# B&R Automation Studio project NAEUL004C00R13L518F00 (part 57)

#### Local.var
```iecst
(*2020-05-26*)
(**)
(*Local Action, State & Status*)
VAR
	eAct : ePullerPusherAction := PPActIdle;
	eStat : ePullerPusherAction := PPActIdle;
	eMainStatus : eFBStatus := Idle;
	eStatus : eFBStatus := Idle;
	eStatus1 : eFBStatus := Idle;
	eStatus2 : eFBStatus := Idle;
	eStatus3 : eFBStatus := Idle;
	udiStatus : UDINT := 0;
	udiStatus1 : UDINT := 0;
	udiStatus2 : UDINT := 0;
	udiStatus3 : UDINT := 0;
	sStatTxt : STRING[200] := '';
	a_sStatText : ARRAY[0..50] OF STRING[200] := ['Idling','Going Width','Full Homing','Powering On','Powering Off','Homing','Moving Absolute','Moving Relative','Jogging Open','Jogging Close','Jogging Stop','Resetting Axis Error','Stopping','Writing SDO','Background Starting Module OK Check','Background Stopping Module OK Check','Going Width And Power Off','Reset Servo Module Node',33('')];
END_VAR
(**)
(*Local Alarm*)
VAR
	tyAlmData : tyAlmDat;
	tyAlmData1 : tyAlmDat;
	tyAlmData2 : tyAlmDat;
	tyAlmData3 : tyAlmDat;
	a_tyAlmText : ARRAY[10000..10299] OF tyAlmTxt := [(sAlmText:='Axis Move Abnormally By External Force',sRcyText:='Servo Motor Abnormal Operation. Reset And Resume Operation. If The Problem Persists, Please Contact Nutek For A Possible Solution.'),(sAlmText:='CANOpen Communication Error, ModuleOK Not TRUE',sRcyText:='Fail While Read/Write Data. Reset The Error And Resume Operation.'),(sAlmText:='Power On Time Out While Going New Width',sRcyText:='Timeout Expired Before Operation Completed. Reset And Resume Operation.'),(sAlmText:='Homing Time Out While Going New Width',sRcyText:='Timeout Expired Before Operation Completed. Reset And Resume Operation.'),(sAlmText:='Move Absolute Time Out While Going New Width',sRcyText:='Timeout Expired Before Operation Completed. Reset And Resume Operation.'),(sAlmText:='Stop Motion Time Out While Going New Width',sRcyText:='Timeout Expired Before Operation Completed. Reset And Resume Operation.'),(sAlmText:='Axis Error Reset Failed While Going New Width',sRcyText:='Axis Error Reset Failed. Please Retry Again Reset Operation. If The Problem Persists, Please Contact Nutek For A Possible Solution.'),(sAlmText:='Axis Error Occur In Move Absolute While Going New Width',sRcyText:='Servo Motor Abnormal Operation. Reset And Resume Operation. If The Problem Persists, Please Contact Nutek For A Possible Solution.'),(sAlmText:='Axis Error Occur In Homing While Going New Width',sRcyText:='Servo Motor Abnormal Operation. Reset And Resume Operation. If The Problem Persists, Please Contact Nutek For A Possible Solution.'),(sAlmText:='Homing Done But Home Flag Is Not Activated While Going New Width',sRcyText:='Servo Motor Abnormal Operation. Reset And Resume Operation. If The Problem Persists, Please Contact Nutek For A Possible Solution.'),(sAlmText:='Forward Limit Activated In Homing While Going New Width',sRcyText:='Forward Limit Switch Is Activated. Reset The Error By Operate The Motor Backwards.'),(sAlmText:='Reverse Limit Activated In Homing While Going New Width',sRcyText:='Reverse Limit Switch Is Activated. Reset The Error By Operate The Motor Backwards.'),(sAlmText:='Forward Limit Activated In Move Absolute While Going New Width',sRcyText:='Forward Limit Switch Is Activated. Reset The Error By Operate The Motor Backwards.'),(sAlmText:='Reverse Limit Activated In Move Absolute While Going New Width',sRcyText:='Reverse Limit Switch Is Activated. Reset The Error By Operate The Motor Backwards.'),(sAlmText:='Power On Time Out While Full Homing',sRcyText:='Timeout Expired Before Operation Completed. Reset And Resume Operation.'),(sAlmText:='Homing Time Out While Full Homing',sRcyText:='Timeout Expired Before Operation Completed. Reset And Resume Operation.'),(sAlmText:='Stop Motion Time Out While Full Homing',sRcyText:='Timeout Expired Before Operation Completed. Reset And Resume Operation.'),(sAlmText:='Axis Error Reset Failed While Full Homing',sRcyText:='Axis Error Reset Failed. Please Retry Again Reset Operation. If The Problem Persists, Please Contact Nutek For A Possible Solution.'),(sAlmText:='Axis Error Occur In Homing While Full Homing',sRcyText:='Servo Motor Abnormal Operation. Reset And Resume Operation. If The Problem Persists, Please Contact Nutek For A Possible Solution.'),(sAlmText:='Homing Done But Home Flag Is Not Activated While Full Homing',sRcyText:='Servo Motor Abnormal Operation. Reset And Resume Operation. If The Problem Persists, Please Contact Nutek For A Possible Solution.'),(sAlmText:='Forward Limit Activated In Homing While Full Homing',sRcyText:='Forward Limit Switch Is Activated. Reset The Error By Operate The Motor Backwards.'),(sAlmText:='Reverse Limit Activated In Homing While Full Homing',sRcyText:='Reverse Limit Switch Is Activated. Reset The Error By Operate The Motor Backwards.'),(sAlmText:='Power On Time Out',sRcyText:='Timeout Expired Before Operation Completed. Reset And Resume Operation.'),(sAlmText:='Power Off Time Out',sRcyText:='Timeout Expired Before Operation Completed. Reset And Resume Operation.'),(sAlmText:='Homing Time Out',sRcyText:='Timeout Expired Before Operation Completed. Reset And Resume Operation.'),(sAlmText:='Move Absolute Time Out',sRcyText:='Timeout Expired Before Operation Completed. Reset And Resume Operation.'),(sAlmText:='Move Relative Time Out',sRcyText:='Timeout Expired Before Operation Completed. Reset And Resume Operation.'),(sAlmText:='Stop Motion Time Out',sRcyText:='Timeout Expired Before Operation Completed. Reset And Resume Operation.'),(sAlmText:='SDO Write Error',sRcyText:='Fail While Write Data. Reset The Error And Resume Operation.'),(sAlmText:='Request Absolute Position Out Of Range',sRcyText:='Request Absolute Position Does Not Fall Within The Expected Range.'),(sAlmText:='Inlet Sensor Interrupt Auto Width Movement',sRcyText:='Operation Stop Due To The Interruption Of Sensor While Auto Width Moving. Solve The Interruption To Resume Operation.'),(sAlmText:='Outlet Sensor Interrupt Auto Width Movement',sRcyText:='Operation Stop Due To The Interruption Of Sensor While Auto Width Moving. Solve The Interruption To Resume Operation.'),(sAlmText:='Clear Sensor Interrupt Auto Width Movement',sRcyText:='Operation Stop Due To The Interruption Of Sensor While Auto Width Moving. Solve The Interruption To Resume Operation.'),(sAlmText:='Middle Sensor Interrupt Auto Width Movement',sRcyText:='Operation Stop Due To The Interruption Of Sensor While Auto Width Moving. Solve The Interruption To Resume Operation.'),(sAlmText:='Sensor Interrupt Auto Width Movement',sRcyText:='Operation Stop Due To The Interruption Of Sensor While Auto Width Moving. Solve The Interruption To Resume Operation.'),(sAlmText:='Power On Time Out While Going New Width And Off',sRcyText:='Timeout Expired Before Operation Completed. Reset And Resume Operation.'),(sAlmText:='Homing Time Out While Going New Width And Off',sRcyText:='Timeout Expired Before Operation Completed. Reset And Resume Operation.'),(sAlmText:='Move Absolute Time Out While Going New Width And Off',sRcyText:='Timeout Expired Before Operation Completed. Reset And Resume Operation.'),(sAlmText:='Stop Motion Time Out While Going New Width And Off',sRcyText:='Timeout Expired Before Operation Completed. Reset And Resume Operation.'),(sAlmText:='Axis Error Reset Failed While Going New Width And Off',sRcyText:='Axis Error Reset Failed. Please Retry Again Reset Operation. If The Problem Persists, Please Contact Nutek For A Possible Solution.'),(sAlmText:='Axis Error Occur In Move Absolute While Going New Width And Off',sRcyText:='Servo Motor Abnormal Operation. Reset And Resume Operation. If The Problem Persists, Please Contact Nutek For A Possible Solution.'),(sAlmText:='Axis Error Occur In Homing While Going New Width And Off',sRcyText:='Servo Motor Abnormal Operation. Reset And Resume Operation. If The Problem Persists, Please Contact Nutek For A Possible Solution.'),(sAlmText:='Homing Done But Home Flag Is Not Activated While Going New Width And Off',sRcyText:='Servo Motor Abnormal Operation. Reset And Resume Operation. If The Problem Persists, Please Contact Nutek For A Possible Solution.'),(sAlmText:='Forward Limit Activated In Homing While Going New Width And Off',sRcyText:='Forward Limit Switch Is Activated. Reset The Error By Operate The Motor Backwards.'),(sAlmText:='Reverse Limit Activated In Homing While Going New Width And Off',sRcyText:='Reverse Limit Switch Is Activated. Reset The Error By Operate The Motor Backwards.'),(sAlmText:='Forward Limit Activated In Move Absolute While Going New Width And Off',sRcyText:='Forward Limit Switch Is Activated. Reset The Error By Operate The Motor Backwards.'),(sAlmText:='Reverse Limit Activated In Move Absolute While Going New Width And Off',sRcyText:='Reverse Limit Switch Is Activated. Reset The Error By Operate The Motor Backwards.'),2((sAlmText:='Sensor Interrupt Auto Width Movement',sRcyText:='Operation Stop Due To The Interruption Of Sensor While Auto Width Moving. Solve The Interruption To Resume Operation.')),249((0)),(sAlmText:='Forward Limit Activated',sRcyText:='Forward Limit Switch Is Activated. Reset The Error By Operate The Motor Backwards.'),(sAlmText:='Reverse Limit Activated',sRcyText:='Reverse Limit Switch Is Activated. Reset The Error By Operate The Motor Backwards.')];
END_VAR
(**)
(*Local Output*)
VAR
	tyParamOut : tyMotionCANParamOut;
	sAxisErrTxt : STRING[80];
	bWidthPosDiff : BOOL;
	bJogOpen : BOOL;
	bJogClose : BOOL;
	bJogging : BOOL;
	bOpenSen : BOOL;
	bCloseSen : BOOL;
END_VAR
(**)
(*Local Input*)
VAR
	udiRstErr : UDINT := 0;
	bPrep : BOOL := TRUE;
	bEn : BOOL := TRUE;
	bDis : BOOL := FALSE;
	bOps : BOOL := FALSE;
	bManual : BOOL := FALSE;
	diWidthAtHmPos : DINT := 400;
	tyTuning : tyMotionCANTuning;
	diGoWidth : DINT := 150;
	diJogVelInUMPS : DINT := 10000;
	diMovePosInUM : DINT := 0;
	diMoveDistInUM : DINT := 0;
	diMoveVelInUMPS : DINT := 10000;
	diMoveAcc : DINT := 500;
	diMoveDec : DINT := 500;
	diMinAbsPosInUM : DINT := -3000;
	diMaxAbsPosInUM : DINT := 10000000;
	diMinWidthInUM : DINT := 70000;
	diMaxWidthInUM : DINT := 460000;
	diWidthOffsetInUM : DINT := 0;
	bInletSensor : BOOL;
	bOutletSensor : BOOL;
	bClearSensor : BOOL;
	bMiddleSensor : BOOL;
	bInterruptSensor : BOOL;
	bOpenInterruptSensor : BOOL;
	bCloseInterruptSensor : BOOL;
	bDir : BOOL;
	bDirBl : BOOL;
	bNoIndexPulse : BOOL;
	usiNode : USINT;
	sDevice : STRING[3];
	sProgNm : STRING[15] := 'AWOpen';
	diMoveBacklashDistInUM : DINT := 3000;
	diPitchInUM : DINT := 3000;
	tyParamInHm : tyMotionCANParamInHm;
	tyParamInConvert : tyMotionCANParamInConvert := (diPitchInUM:=3000);
	bNtSettingsLoadDone : BOOL := TRUE;
	eMotorType : eServoMotorType := DeltaAsdaA2;
	usiJogFwdStep : USINT;
	usiJogRevStep : USINT;
	bJogRevDone : BOOL;
	bJogFwdDone : BOOL;
	bJogStopDone : BOOL;
	bJogFwd : BOOL;
	bJogRev : BOOL;
	diServoTorque : DINT := 100;
	udiMaxTorque : UDINT := 100;
	diRetSpd : DINT := 24000;
END_VAR
(**)
(*Local*)
VAR
	bRstErr : BOOL;
	udiRstErrOld : UDINT;
	bInitDone : BOOL;
	bInitialDone : BOOL;
	bModuleOKChk : BOOL := TRUE;
	bModuleOK : BOOL;
	bModuleNotOK : BOOL := TRUE;
	diMtrPshrExtTrq : DINT := 0;
	bModuleNotOKLock : BOOL;
	bNotInterruptible : BOOL;
	bInterruptSensor1 : BOOL;
	bInterruptSensor2 : BOOL;
	diActualPosInUMOld : DINT;
	diSlowSpeed : DINT := 2800;
	diExtSlowSpeed : DINT := 2800;
	usiRstStep : USINT := 0;
	usiStep : USINT;
	usiCount : USINT;
	fbTm : TON := (PT:=T#2s);
	fbServoModuleNotOk : TON := (IN:=FALSE,PT:=T#2s);
	fbServoModuleOk : TON := (IN:=FALSE,PT:=T#5s);
	fbRstNodeTimer : TON := (PT:=T#3s);
	tyParamInMove : tyMotionCANParamInMove;
	tyParamInDriver : tyMotionCANDriverIn;
	tyParamOutDriver : tyMotionCANDriverOut := (siModOfOpt_6060:=6);
	fbStop : fbMotionCANStop;
	fbRstAxisErr : fbMotionCANRstAxisErr;
	fbJog : fbMotionCANJog;
	fbMovRel : fbMotionCANMovRel;
	fbMovAbs : fbMotionCANMovAbs;
	fbHoming : fbMotionCANHoming;
	fbPwrOff : fbMotionCANPwrOff;
	fbPwrOn : fbMotionCANPwrOn;
	fbFullHm : fbMotionCANFullHm;
	fbFullMovAbs : fbMotionCANFullMovAbs;
	fbFullMovAbsBl : fbMotionCANFullMovAbsBl;
	fbModuleOK : fbMotionCANModuleOK;
	fbSDOWrite : fbCANSDOWriteArrayParam;
	fbSDOWriteTorque : CANopenSDOWrite8;
	udiModuleNum : UDINT := 301;
END_VAR
```

#### Act_Action.st
```iecst
(** 2020-03-16 **)
ACTION Act_Action:

	//Reset Error
	IF (eStatus = Error) AND bRstErr THEN
		p_eAct	:= PPActIdle;
		eStat	:= PPActIdle;

		fMotionCANRstCtrlWord(ADR(tyParamOutDriver));
	END_IF

	//Reset Done
	IF eStatus = Done AND p_eAct = PPActIdle THEN
		eStat	:= PPActIdle;
	END_IF

	//Set p_eAct
	IF (eStatus = Idle
		AND eStatus1 = Idle
		AND eStatus2 = Idle
		AND eStatus3 = Idle)
		OR p_eAct = PPActIdle
		OR p_eAct = PPActStop
		OR (p_eAct = PPActJogStop AND eStatus = Done)
		THEN
		eStat	:= p_eAct;
	END_IF

	IF EDGEPOS(bModuleNotOK) THEN
		eStat := PPActIdle;
	END_IF

END_ACTION
```

#### Act_Alarm.st
```iecst
(** 2020-03-16 **)
ACTION Act_Alarm:

	//Error
	IF EDGEPOS(eStatus = Error) THEN

		tyAlmData.sProgNm		:= p_sProgNm;
		tyAlmData.udiCode		:= udiStatus;
		tyAlmData.eSeverity		:= AlmSeverityError;
		tyAlmData.udiRunTime	:= tyAlmData.udiRunTime + 1;
		tyAlmData.bAlm			:= TRUE;
		tyAlmData.udiModuleNum  := udiModuleNum;
		g_sAWCloseProgNm		:= p_sProgNm;
		//Get Error Message
		IF tyAlmData.udiCode < 10000 OR tyAlmData.udiCode > 10299 THEN
			tyAlmData.sAlmMsg	:= 'Unknown';
			tyAlmData.sRcyMsg	:= 'Unknown';
		ELSE
			tyAlmData.sAlmMsg	:= a_tyAlmText[tyAlmData.udiCode].sAlmText;
			tyAlmData.sRcyMsg	:= a_tyAlmText[tyAlmData.udiCode].sRcyText;
		END_IF

		sStatTxt	:= tyAlmData.sAlmMsg;

	ELSIF bRstErr AND (tyAlmData.udiCode <> 0) THEN

		tyAlmData.udiCode	:= 0;
		tyAlmData.eSeverity	:= AlmSeverityNA;
		tyAlmData.sAlmMsg	:= '';
		tyAlmData.sRcyMsg	:= '';
		tyAlmData.bAlm			:= FALSE;
		sStatTxt	:= a_sStatText[eStat];

	END_IF

END_ACTION
```

#### Act_Alarm1.st
```iecst
(** 2020-03-16 **)
ACTION Act_Alarm1:

	//Error
	IF EDGEPOS(eStatus1 = Error) THEN

		tyAlmData1.sProgNm		:= p_sProgNm;
		tyAlmData1.udiCode		:= udiStatus1;
		tyAlmData1.eSeverity	:= AlmSeverityError;
		tyAlmData1.udiRunTime	:= tyAlmData1.udiRunTime + 1;
		tyAlmData1.bAlm			:= TRUE;
		tyAlmData1.udiModuleNum  := udiModuleNum;
		g_sAWCloseProgNm		:= p_sProgNm;
		//Get Error Message
		IF tyAlmData1.udiCode < 10000 OR tyAlmData1.udiCode > 10099 THEN
			tyAlmData1.sAlmMsg	:= 'Unknown';
			tyAlmData1.sRcyMsg	:= 'Unknown';
		ELSE
			tyAlmData1.sAlmMsg	:= a_tyAlmText[tyAlmData1.udiCode].sAlmText;
			tyAlmData1.sRcyMsg	:= a_tyAlmText[tyAlmData1.udiCode].sRcyText;
		END_IF

		sStatTxt	:= tyAlmData1.sAlmMsg;

	ELSIF bRstErr AND (tyAlmData1.udiCode <> 0) THEN

		tyAlmData1.udiCode		:= 0;
		tyAlmData1.eSeverity	:= AlmSeverityNA;
		tyAlmData1.sAlmMsg		:= '';
		tyAlmData1.sRcyMsg		:= '';
		tyAlmData1.bAlm			:= FALSE;
		sStatTxt	:= a_sStatText[eStat];

	END_IF

END_ACTION
```

#### Act_Alarm2.st
```iecst
(** 2020-03-16 **)
ACTION Act_Alarm2:

	//Error
	IF EDGEPOS(eStatus2 = Error) THEN

		tyAlmData2.sProgNm		:= p_sProgNm;
		tyAlmData2.udiCode		:= udiStatus2;
		tyAlmData2.eSeverity	:= AlmSeverityError;
		tyAlmData2.udiRunTime	:= tyAlmData2.udiRunTime + 1;
		tyAlmData2.bAlm			:= TRUE;
		tyAlmData2.udiModuleNum  := udiModuleNum;
		g_sAWCloseProgNm		:= p_sProgNm;
		//Get Error Message
		IF tyAlmData2.udiCode < 10000 OR tyAlmData2.udiCode > 10099 THEN
			tyAlmData2.sAlmMsg	:= 'Unknown';
			tyAlmData2.sRcyMsg	:= 'Unknown';
		ELSE
			tyAlmData2.sAlmMsg	:= a_tyAlmText[tyAlmData2.udiCode].sAlmText;
			tyAlmData2.sRcyMsg	:= a_tyAlmText[tyAlmData2.udiCode].sRcyText;
		END_IF

		sStatTxt	:= tyAlmData2.sAlmMsg;

	ELSIF bRstErr AND (tyAlmData2.udiCode <> 0) THEN

		tyAlmData2.udiCode		:= 0;
		tyAlmData2.eSeverity	:= AlmSeverityNA;
		tyAlmData2.sAlmMsg		:= '';
		tyAlmData2.sRcyMsg		:= '';
		tyAlmData2.bAlm			:= FALSE;
		sStatTxt	:= a_sStatText[eStat];

	END_IF

END_ACTION
```

#### Act_Alarm3.st
```iecst
(** 2020-03-16 **)
ACTION Act_Alarm3:

	//Error
	IF EDGEPOS(eStatus3 = Error) THEN

		tyAlmData3.sProgNm		:= p_sProgNm;
		tyAlmData3.udiCode		:= udiStatus3;
		tyAlmData3.eSeverity	:= AlmSeverityError;
		tyAlmData3.udiRunTime	:= tyAlmData3.udiRunTime + 1;
		tyAlmData3.bAlm			:= TRUE;
		tyAlmData3.udiModuleNum  := udiModuleNum;
		g_sAWCloseProgNm		:= p_sProgNm;
		//Get Error Message
		IF tyAlmData3.udiCode < 10000 OR tyAlmData3.udiCode > 10099 THEN
			tyAlmData3.sAlmMsg	:= 'Unknown';
			tyAlmData3.sRcyMsg	:= 'Unknown';
		ELSE
			tyAlmData3.sAlmMsg	:= a_tyAlmText[tyAlmData3.udiCode].sAlmText;
			tyAlmData3.sRcyMsg	:= a_tyAlmText[tyAlmData3.udiCode].sRcyText;
		END_IF

		sStatTxt	:= tyAlmData3.sAlmMsg;

	ELSIF bRstErr AND (tyAlmData3.udiCode <> 0) THEN

		tyAlmData3.udiCode		:= 0;
		tyAlmData3.eSeverity	:= AlmSeverityNA;
		tyAlmData3.sAlmMsg		:= '';
		tyAlmData3.sRcyMsg		:= '';
		tyAlmData3.bAlm			:= FALSE;
		sStatTxt	:= a_sStatText[eStat];

	END_IF

END_ACTION
```

#### Act_Background.st
```iecst
(** 2020-05-26 **)
ACTION Act_Background:

	//Update Parameter
	IF bModuleOK = TRUE THEN

		tyParamInMove.diPosInUM		:= p_diMovePosInUM;
		tyParamInMove.diDistInUM	:= p_diMoveDistInUM;
		tyParamInMove.diVelInUMPS	:= p_diMoveVelInUMPS;
		tyParamInMove.diAcc			:= p_diMoveAcc;
		tyParamInMove.diDec			:= p_diMoveDec;

		fMotionCANUpdtDat(ADR(tyParamOut) , p_tyParamInConvert , tyParamOutDriver , tyParamInDriver , tyParamInMove , p_tyParamInHm , p_bDir, p_eNtParamMotorType);

		bWidthPosDiff	:= (tyParamOut.bIsHomed = FALSE) OR ((ABS((fAWWidthToPosInUM(p_diGoWidth , p_diWidthAtHmPos)) - tyParamOut.diActualPosInUM)) > 500);

		p_tyParamInConvert.diPitchInUM	:= fPitchCalc(p_diWidthOffsetInUM , p_diMaxWidthInUM , p_diMinWidthInUM , p_diPitchInUM);

		fbFullMovAbsBl.tyParamInConvert					:= p_tyParamInConvert;

		IF p_bDir = TRUE THEN
			bOpenSen	:= tyParamOut.bFwdLmtSen;
			bCloseSen	:= tyParamOut.bRevLmtSen;
		ELSE
			bOpenSen	:= tyParamOut.bRevLmtSen;
			bCloseSen	:= tyParamOut.bFwdLmtSen;
		END_IF

		CASE p_eNtParamMotorType OF
			DeltaAsdaA2:
				CASE tyParamOut.udiAxisErrID OF
					8976:	sAxisErrTxt	:= 'Over Current';
					12560:	sAxisErrTxt	:= 'Over Voltage';
					12576:	sAxisErrTxt	:= 'Under Voltage';
					12592:	sAxisErrTxt	:= 'Input Power Phase Loss';
					12816:	sAxisErrTxt	:= 'Regeneration Error';
					12848:	sAxisErrTxt	:= 'Overload';
					12849:	sAxisErrTxt	:= 'Pre-overload Warning';
					13056:	sAxisErrTxt	:= 'U,V,W Wiring Error';
					16912:	sAxisErrTxt	:= 'IGBT Temperature Error';
					21296:	sAxisErrTxt	:= 'Memory Error';
					21569:	sAxisErrTxt	:= 'Emergency Stop Activated';
					21570:	sAxisErrTxt	:= 'Forward Limit Switch Error';
					21571:	sAxisErrTxt	:= 'Reverse Limit Switch Error';
					21572:	sAxisErrTxt	:= 'Forward Software Limit';
					21573:	sAxisErrTxt	:= 'Reverse Software Limit';
					21760:	sAxisErrTxt	:= 'DSP Firmware Upgrade';
					25088:	sAxisErrTxt	:= 'CANopen SYNC Error';
					25360:	sAxisErrTxt	:= 'CANopen Data Initial Error';
					25376:	sAxisErrTxt	:= 'Adjustment Error';
					28961:	sAxisErrTxt	:= 'Motor Protection Error';
					28962:	sAxisErrTxt	:= 'Motor Error';
					29445:	sAxisErrTxt	:= 'Encoder Error';
					29446:	sAxisErrTxt	:= 'Encoder Output Error';
					29968:	sAxisErrTxt	:= 'Serial Communication Error';
					29984:	sAxisErrTxt	:= 'Serial Communication Time Out';
					33024:	sAxisErrTxt	:= 'CANbus Error (Bus-off)';
					33040:	sAxisErrTxt	:= 'CANopen SDO receive buffer overrun';
					33056:	sAxisErrTxt	:= 'CANbus Error (Warning)';
					33072:	sAxisErrTxt	:= 'Node Guarding or Heartbeat Error';
					33280:	sAxisErrTxt	:= 'CANopen PDO Object Error';
					33792:	sAxisErrTxt	:= 'Over Speed';
					34304:	sAxisErrTxt	:= 'Abnormal Pulse Control Command';
					34320:	sAxisErrTxt	:= 'Full Closed Loop Excessive Deviation';
					34321:	sAxisErrTxt	:= 'Excessive Deviation';
				END_CASE

			SchneiderLexium28:
				CASE tyParamOut.udiAxisErrID OF
					8724:	sAxisErrTxt	:= 'Over Current';
					8976:	sAxisErrTxt	:= 'Motor Overload';
					8977:	sAxisErrTxt	:= 'Drive overload (foldback)';
					9088:	sAxisErrTxt	:= 'Calculated offsets for current sensors out OF range';
					9089:	sAxisErrTxt := 'Motor phase missing';
					9090:	sAxisErrTxt := 'Overcurrent detected at one OF the digital outputs';
					12560:	sAxisErrTxt	:= 'DC Bus Over Voltage';
					12576:	sAxisErrTxt	:= 'DC Bus Under Voltage';
					12672:	sAxisErrTxt	:= 'Braking Resistor Overload';
					12673:	sAxisErrTxt	:= 'Safety function Safe Torque Off (STO) triggered';
					12674:	sAxisErrTxt	:= 'DC bus voltage measurement';
					12675:	sAxisErrTxt	:= 'Missing mains supply, undervoltage mains supply';
					12676:	sAxisErrTxt := 'The encoder supply voltage has dropped under operational value';
					12677:	sAxisErrTxt := 'The multi turn encoder battery voltage has dropped under 3 Vdc';
					12678:	sAxisErrTxt := 'Internal position synchronization error	detected between the multi turn AND the single turn modules';
					12679:	sAxisErrTxt := 'Generic error code of the multi turn module is detected';
					12697:	sAxisErrTxt := 'Braking resistor overload';
					16512:	sAxisErrTxt	:= 'Drive overtemperature (IPM)';
					16513:	sAxisErrTxt	:= 'Drive overtemperature (controller)';
					16534:	sAxisErrTxt := 'Temperature sensor inoperative';
					17168:	sAxisErrTxt	:= 'Power stage overtemperature';
					17280:	sAxisErrTxt := 'The encoder temperature is too high';
					17424:	sAxisErrTxt	:= 'Motor overtemperature';
					21808:	sAxisErrTxt	:= 'System error detected (nonvolatilememory)';
					21893:	sAxisErrTxt	:= 'Error detected in non-volatile memory';
					21889:	sAxisErrTxt	:= 'System error detected (nonvolatile memory)';
					21890:	sAxisErrTxt	:= 'System error detected (CAN power supply)';
					21891:	sAxisErrTxt	:= 'System error detected (selftest)';
					21894:	sAxisErrTxt	:= 'System error detected (NV ACCESS)';
					25472:	sAxisErrTxt	:= 'Target position rejected';
					25985:	sAxisErrTxt	:= 'System error detected(FPGA)';
					28816:	sAxisErrTxt	:= 'System error detected (FPGA does NOT match firmware)';
					28817:	sAxisErrTxt	:= 'Emergency Stop Activated';
					28961:	sAxisErrTxt := 'Motor blocked';
					29080:	sAxisErrTxt := 'Commutation error detected';
					29568:  sAxisErrTxt	:= 'Error detected in communication with motor encoder';
					29574:	sAxisErrTxt	:= 'Drive is not synchronous wit master cycle';
					29581:	sAxisErrTxt := 'System error detected (encoder)';
					29587:	sAxisErrTxt	:= 'Encoder overvoltage or overcurrent';
					29592:	sAxisErrTxt := 'The returned position value are no longer considered valid';
					29593:	sAxisErrTxt := 'The multi turn encoder requires an explicit configuration command';
					30081:	sAxisErrTxt := 'Target position rejected';
					30082:	sAxisErrTxt := 'No target values received via the fieldbus';
					33072:	sAxisErrTxt	:= 'CANopen: Heartbeat error detected';
					33296:	sAxisErrTxt := 'R_PDO is too short';
					33921:	sAxisErrTxt	:= 'Actual Motor Velocity Too High';
					33553:	sAxisErrTxt	:= 'Motor torque too high FOR an excessive period OF time';
					33664:	sAxisErrTxt := 'Unstable current loop';
					33922:	sAxisErrTxt := 'Velocity deviation too high';
					34321:	sAxisErrTxt	:= 'Position deviation too high';
					34432:	sAxisErrTxt := 'Position deviation via signal output function MC_OK';
					34441:	sAxisErrTxt := 'Position deviation too high (following error)';
					61568:	sAxisErrTxt	:= 'Fieldbus: Communication	error detected';
					65282:	sAxisErrTxt	:= 'Not possible to read data of electronic motor nameplate';
					65296:	sAxisErrTxt	:= 'Forward Limit Switch Error';
					65297:	sAxisErrTxt	:= 'Reverse Limit Switch Error';
					65281:	sAxisErrTxt := 'System error detected';
					65298:	sAxisErrTxt	:= 'Forward Software Limit';
					65299:	sAxisErrTxt	:= 'Reverse Software Limit';
					65301:	sAxisErrTxt := 'The encoder firmware cannot operate on the provided hardware';

				END_CASE

			EstunPronet:
				CASE tyParamOut.udiAxisErrID OF
					65281:	sAxisErrTxt	:= 'Parameter breakdown';//A01
					65282:	sAxisErrTxt	:= 'AD shift channels breakdown';
					65283:	sAxisErrTxt	:= 'Overspeed';
					65284:	sAxisErrTxt	:= 'Overload';
					65285:	sAxisErrTxt := 'Position error counteroverflow ';
					65286:	sAxisErrTxt := 'Position error pulse overflow';
					65287:	sAxisErrTxt	:= 'The setting of electronic gear or given pulse frequency is not reasonable';
					65288:	sAxisErrTxt	:= 'The 1st channel of current detection is wrong.';
					65289:	sAxisErrTxt	:= 'The 2nd channel of current detection is wrong.';
					65290:	sAxisErrTxt	:= 'Incremental Encoder is break off.';//A10
					65292:	sAxisErrTxt	:= 'Overcurrent';
					65293:	sAxisErrTxt	:= 'Overvoltage';
					65294:	sAxisErrTxt	:= 'Undervoltage';
					65295:	sAxisErrTxt := 'Bleeder resistor error';
					65296:	sAxisErrTxt := 'Regeneration error';
					65297:	sAxisErrTxt := 'Resolver error';
					65298:	sAxisErrTxt := 'IGBT superheat alarm';
					65299:	sAxisErrTxt := 'Motor overheat alarm';
					65300:	sAxisErrTxt := 'Power line phase shortage';//A20
					65301:	sAxisErrTxt	:= 'Instantaneous power off alarm';
					65302:	sAxisErrTxt	:= 'Motor temperature detection sensor is break off.';
					65303:	sAxisErrTxt := 'Brake overcurrent alarm';//A23
					65305:	sAxisErrTxt := 'Motor power line U overcurrent';//A25
					65306:	sAxisErrTxt := 'Motor power line V overcurrent';//A26
					65307:	sAxisErrTxt := 'Motor power line W overcurrent';//A27
					65322:	sAxisErrTxt	:= 'Servomotor type error';//A42
					65323:	sAxisErrTxt	:= 'Servo drive type error';
					65325:	sAxisErrTxt	:= 'Absolute encoder multiturn information error';
					65326:	sAxisErrTxt	:= 'Absolute encoder multiturn information overflow';
					65327:	sAxisErrTxt	:= 'Battery voltage below 2.5V';
					65328:	sAxisErrTxt	:= 'Battery voltage below 3.1V';//A48
					65330:	sAxisErrTxt := 'Serial encoder communication overtime ';//A50
					65331:	sAxisErrTxt := 'Absolute encoder overspeed alarm detected';
					65332:  sAxisErrTxt	:= 'Absolute state of serial encoder error';
					65333:	sAxisErrTxt	:= 'Serial encoder calcaution error';
					65334:	sAxisErrTxt := 'Parity bit or end bit in serial encoder control domain error';
					65335:	sAxisErrTxt	:= 'Serial encoder communication data checking error';
					65336:	sAxisErrTxt := 'End bit in serial encoder control domain error';
					65338:	sAxisErrTxt := 'Serial encoder data empty';
					65339:	sAxisErrTxt := 'Serial encoder data format error';
					65340:	sAxisErrTxt := 'Communication module not detected ';//A60
					65341:	sAxisErrTxt := 'Communication unsuccessful';
					65342:	sAxisErrTxt := 'Servo drive can not receive the period data of communication module ';
					65343:	sAxisErrTxt := 'Communication module can not receive the servo drive response data.';
					65344:	sAxisErrTxt := 'Communication module and bus connectionless';
					65346:	sAxisErrTxt := 'CAN communication abnormal';
					65347:	sAxisErrTxt := 'Receiving heartbeat timeout';
					65349:	sAxisErrTxt := 'Synchronization signal monitoring cycle is longer than setting';
					65362: sAxisErrTxt	:= 'Torque output alarm';
				END_CASE
		END_CASE

	ELSE

		tyParamOut.bAxisErr			:= FALSE;
		tyParamOut.bFwdLmtSen		:= FALSE;
		tyParamOut.bInPos			:= FALSE;
		tyParamOut.bIsHomed			:= FALSE;
		tyParamOut.bPosDiff			:= TRUE;
		tyParamOut.bPwrOn			:= FALSE;
		tyParamOut.bRevLmtSen		:= FALSE;
		tyParamOut.bStopped			:= TRUE;
		tyParamOut.diActualPosInUM	:= 0;
		tyParamOut.diHmAcc			:= 0;
		tyParamOut.diHmSpdForSwitch	:= 0;
		tyParamOut.diHmSpdForZero	:= 0;
		tyParamOut.diProfileAcc		:= 0;
		tyParamOut.diProfileDec		:= 0;
		tyParamOut.udiAxisErrID		:= 0;

		bWidthPosDiff				:= TRUE;

	END_IF

	//Abnormal Movement
//	IF eStatus1 <> Error THEN
//		IF p_bOps = TRUE AND eStatus = Idle THEN
//			IF (ABS(tyParamOut.diActualPosInUM - diActualPosInUMOld) > 2000) AND (ABS(tyParamOut.diActualPosInUM - diActualPosInUMOld) < 10000) THEN
//				eStatus1	:= Error;
//				udiStatus1	:= 10000;	//Axis Move Abnormally By External Force
//
//				fMotionCANRstCtrlWord(ADR(tyParamOutDriver));
//				p_eAct	:= PPActIdle;
//				eStat	:= PPActIdle;
//			END_IF
//		ELSE
//			diActualPosInUMOld	:= tyParamOut.diActualPosInUM;
//		END_IF
//	END_IF

	//Reset Error
	IF (eStatus1 = Error) AND bRstErr THEN
		eStatus1	:= Idle;
		udiStatus1	:= 0;
	END_IF

	//Request Position To Movement Out Of Range
	IF p_bOps
		AND((tyParamInMove.diPosInUM < p_diMinAbsPosInUM) OR (tyParamInMove.diPosInUM > p_diMaxAbsPosInUM))
		AND (eStatus2 <> Error) THEN
		eStatus2	:= Error;
		udiStatus2	:= 10029;	//Request Absolute Position Out Of Range

		fMotionCANRstCtrlWord(ADR(tyParamOutDriver));
		p_eAct	:= PPActIdle;
		eStat	:= PPActIdle;
	END_IF

	//Reset Error
	IF (eStatus2 = Error) AND bRstErr THEN
		eStatus2	:= Idle;
		udiStatus2	:= 0;
	END_IF

	//Sensor Interrupt
	IF (bNotInterruptible = TRUE OR bJogging) AND eStatus3 <> Error THEN

		IF p_bInletSensor = TRUE THEN
			eStatus3	:= Error;
			udiStatus3	:= 10030;	//Inlet Sensor Interrupt Auto Width Movement

			fMotionCANRstCtrlWord(ADR(tyParamOutDriver));
			p_eAct	:= PPActIdle;
			eStat	:= PPActIdle;

		ELSIF p_bOutletSensor = TRUE THEN
			eStatus3	:= Error;
			udiStatus3	:= 10031;	//Outlet Sensor Interrupt Auto Width Movement

			fMotionCANRstCtrlWord(ADR(tyParamOutDriver));
			p_eAct	:= PPActIdle;
			eStat	:= PPActIdle;

		ELSIF p_bClearSensor = TRUE THEN
			eStatus3	:= Error;
			udiStatus3	:= 10032;	//Clear Sensor Interrupt Auto Width Movement

			fMotionCANRstCtrlWord(ADR(tyParamOutDriver));
			p_eAct	:= PPActIdle;
			eStat	:= PPActIdle;

		ELSIF p_bMiddleSensor = TRUE THEN
			eStatus3	:= Error;
			udiStatus3	:= 10033;	//Middle Sensor Interrupt Auto Width Movement

			fMotionCANRstCtrlWord(ADR(tyParamOutDriver));
			p_eAct	:= PPActIdle;
			eStat	:= PPActIdle;

		ELSIF p_bInterruptSensor = TRUE THEN
			eStatus3	:= Error;
			udiStatus3	:= 10034;	//Sensor Interrupt Auto Width Movement

			fMotionCANRstCtrlWord(ADR(tyParamOutDriver));
			p_eAct	:= PPActIdle;
			eStat	:= PPActIdle;

		ELSIF p_bCloseInterruptSensor = TRUE AND bJogOpen = FALSE THEN
			eStatus3	:= Error;
			udiStatus3	:= 10047;	//Sensor Interrupt Auto Width Movement

			fMotionCANRstCtrlWord(ADR(tyParamOutDriver));
			p_eAct	:= PPActIdle;
			eStat	:= PPActIdle;

		ELSIF p_bOpenInterruptSensor = TRUE AND bJogClose = FALSE THEN
			eStatus3	:= Error;
			udiStatus3	:= 10048;	//Sensor Interrupt Auto Width Movement

			fMotionCANRstCtrlWord(ADR(tyParamOutDriver));
			p_eAct	:= PPActIdle;
			eStat	:= PPActIdle;
		END_IF

	END_IF

	//Reset Error
	IF (eStatus3 = Error AND bRstErr)
		OR (p_bOpenInterruptSensor AND eStat = PPActJogClose)
		OR (p_bCloseInterruptSensor AND eStat = PPActJogOpen)
		THEN
		eStatus3	:= Idle;
		udiStatus3	:= 0;
	END_IF

	IF bRstErr THEN
		udiStatus	:= 0;
		bJogging	:= FALSE;
		bJogClose	:= FALSE;
		bJogOpen	:= FALSE;
	END_IF

	fbServoModuleOk(IN:= bModuleOK);
	fbServoModuleNotOk(IN:= bModuleOK = FALSE);
	IF fbServoModuleNotOk.Q AND udiStatus <> 10001 THEN

		bModuleNotOK		:= TRUE;
		bModuleNotOKLock	:= TRUE;
		usiRstStep	:= 0;
		tyParamOutDriver.uiCtrlword_6040	:= 0;
		tyParamOutDriver.siModOfOpt_6060	:= 0;
		tyParamOutDriver.diTargetPos_607A	:= 0;
		tyParamOutDriver.udiMoveSpd_6081	:= 0;
		tyParamOutDriver.siHmMethod_6098	:= 0;
		tyParamOutDriver.diJogVel_60FF		:= 0;

		CASE p_eNtParamMotorType OF

			DeltaAsdaA2:
				fbModuleOK(bModuleOK:= FALSE);
				IF eStatus = Idle THEN
					eAct	:= PPActRstNode;
				END_IF

				IF (eStatus = Done OR eStatus = Error)AND eStat = PPActRstNode THEN

					eAct	:= PPActIdle;
				END_IF

			EstunPronet:
				fbModuleOK(bModuleOK:= FALSE);
				IF eStatus = Idle THEN
					eAct	:= PPActRstNode;
				END_IF

				IF (eStatus = Done OR eStatus = Error)AND eStat = PPActRstNode THEN

					eAct	:= PPActIdle;
				END_IF

			SchneiderLexium28:
			// Do Nothing
		END_CASE

	ELSIF bModuleNotOK = TRUE AND fbServoModuleOk.Q THEN

		CASE usiRstStep OF

			0:
				IF eStatus = Idle THEN
					eAct	:= PPActRstAxisErr;
				END_IF

				IF eStatus = Done AND eStat = PPActRstAxisErr THEN
					eAct	:= PPActIdle;
					usiRstStep	:= 4;
				END_IF

			4: tyParamOutDriver.siModOfOpt_6060 := 1;
				usiRstStep	:= 5;

			5: tyParamOutDriver.siModOfOpt_6060 := 1;
				fbRstNodeTimer(IN:=TRUE);

				IF tyParamInDriver.siModOfOptDisp_6061 = 1 THEN
					usiRstStep	:= 6;
					fbRstNodeTimer(IN:=FALSE);
				ELSIF fbRstNodeTimer.Q THEN
					usiRstStep	:= 8;
					fbRstNodeTimer(IN:=FALSE);
				END_IF

			6: tyParamOutDriver.siModOfOpt_6060 := 6;
				fbRstNodeTimer(IN:=FALSE);
				usiRstStep	:= 7;

			7: tyParamOutDriver.siModOfOpt_6060 := 6;
				fbRstNodeTimer(IN:=TRUE);

				IF tyParamInDriver.siModOfOptDisp_6061 = 6 THEN
					usiRstStep	:= 10;
					fbRstNodeTimer(IN:=FALSE);
				ELSIF fbRstNodeTimer.Q THEN
					usiRstStep	:= 9;
					fbRstNodeTimer(IN:=FALSE);
				END_IF

			8:	fbModuleOK(bEn := TRUE, bModuleOK:= FALSE);
				fbRstNodeTimer(IN:=FALSE);
				usiRstStep	:= 9;

			9:	fbModuleOK(bModuleOK:= FALSE);
				IF eStatus = Idle THEN
					eAct	:=PPActRstNode;
				END_IF

				IF eStatus = Done AND eStat = PPActRstNode THEN
					usiRstStep	:= 0;
					eAct		:= PPActIdle;
				END_IF

			10:IF eStatus = Idle THEN
					eAct	:= PPActRstAxisErr;
				END_IF

				IF eStatus = Done AND eStat = PPActRstAxisErr THEN
					eAct			:= PPActIdle;
					usiRstStep	:= 11;
				END_IF

			11:

				IF eStatus = Idle THEN
					eAct	:= PPActSDOWrite;
				END_IF

				IF eStatus = Done AND eStat = PPActSDOWrite THEN
					eAct			:= PPActIdle;
					usiRstStep	:= 13;

				ELSIF udiStatus = 10028 THEN
					eAct			:= PPActIdle;
					usiRstStep	:= 13;
				END_IF

			13: bModuleNotOK	:= FALSE;
				usiRstStep	:= 0;
		END_CASE
	ELSE
		eAct	:= PPActIdle;

	END_IF

	IF tyParamOut.bPosDiff = FALSE THEN
		tyParamOutDriver.uiCtrlword_6040.4	:= FALSE;
	END_IF

END_ACTION
```

#### Act_InitGlobal.st
```iecst
(** 2019-04-09 **)
ACTION Act_InitGlobal:

	(* Always Change If Project Change *)

	//Pass Data To Link
	p_bLinkOpsRun ACCESS p_OpsRun;
	p_bLinkStartupRun ACCESS p_StartupRun;
	p_bLinkPullConvPullerExtCtrl ACCESS p_PshrConvPshrExtCtrl;
	p_bLinkPullConvPullerRetCtrl ACCESS p_PshrConvPshrRetCtrl;
	p_bLinkDIPullerExtRS ACCESS p_DIPusherExtRS;
	p_bLinkDIPullerRetRS ACCESS p_DIPusherRetRS;
	p_bLinkDIPullerExtSlwRS ACCESS p_DIPusherExtSlwSen;
	p_bLinkDIPullerRetSlwRS ACCESS p_DIPusherRetSlwSen;
	p_dintLinkPullerRetSpd ACCESS p_ProdRcpCurrRcp1MtrPshrExtSpd;
	p_dintLinkPullerRetTrq ACCESS p_ProdRcpCurrRcp1MtrPshrExtTorq;

	p_diLinkProdRcpTrq ACCESS p_ProdRcpCurrRcp1MtrPshrExtTorq;
	p_tyLinkTorqParam ACCESS p_NtParamPPTorqParam;

	//Pass Data To Internal Use
	p_udiRstErr ACCESS p_RstErrReset;
	p_bPrep ACCESS p_NtParamProjServoPullPusherPrep;
	p_bOps ACCESS p_OpsStatusRun;
	p_bManual ACCESS p_UIMnlMod;
	p_tyTuning ACCESS p_NtParamPPTuning;
//	p_diJogVelInUMPS ACCESS p_UIMnlPPJogSpd;
	p_diMovePosInUM ACCESS p_UIMnlPPTargetPos;
	p_diMoveDistInUM ACCESS p_UIMnlPPStepSize;
	p_diMoveAcc ACCESS p_NtParamPPAcc;
	p_diMoveDec ACCESS p_NtParamPPDec;
	p_diWidthOffsetInUM ACCESS p_NtParamWidthOffset;
	p_bDir ACCESS p_NtParamPPDir;
	p_bDirBl ACCESS p_NtParamPPDirBl;
	p_usiNode ACCESS p_NtParamPPNode;
	p_sDevice ACCESS p_NtParamPPDevice;
	p_sProgNm ACCESS p_NtParamPPProgNm;
	p_diMoveBacklashDistInUM ACCESS p_NtParamPPMovBlDistInUM;
	p_diPitchInUM ACCESS p_NtParamPPPitchInUM;
	p_tyParamInHm ACCESS p_NtParamPPParamInHm;
	p_tyParamInConvert ACCESS p_NtParamPPParamInConvert;
	p_bNtSettingsLoadDone ACCESS p_StartupNtSettingsLoadDone;
	p_eNtParamMotorType ACCESS p_NtParamPPMotorType;

	p_bInletShutterCloseRS ACCESS p_DIInShutterCloseRS;
	p_bOutletShutterCloseRS ACCESS p_DIOutShutterCloseRS;
	p_bProjInletShutPrep ACCESS p_NtParamProjInletShutPrep;
	p_bProjOutletShutPrep ACCESS p_NtParamProjOutletShutPrep;
	p_bMagWidthChkSen ACCESS p_DIMagWidthChkSen;

	(* Always Change If Project Change *)

END_ACTION
```

#### Act_Initial.st
```iecst
(** 2020-03-16 **)
ACTION Act_Initial:

	//Initial
	sStatTxt	:= a_sStatText[eStat];

	tyParamInMove.diBacklashDistInUM	:= p_diMoveBacklashDistInUM;
	tyParamInMove.diAcc					:= p_diMoveAcc;
	tyParamInMove.diDec					:= p_diMoveDec;

	//p_tyParamInConvert.diPitchInUM	:= fPitchCalc(p_diWidthOffsetInUM , p_diMaxWidthInUM , p_diMinWidthInUM , p_diPitchInUM);

	fbModuleOK.sDevice	:= p_sDevice;
	fbModuleOK.usiNode	:= p_usiNode;
	fbModuleOK.tDlyTm	:= T#5s;
	fbModuleOK(bEn := FALSE);

	fbSDOWrite.sDevice		:= p_sDevice;
	fbSDOWrite.usiNode		:= p_usiNode;
	fbSDOWrite.eMotorType	:= p_eNtParamMotorType;
	fbSDOWrite(bEn := FALSE);

	fbFullMovAbsBl.p_tyParamOutDriver				:= ADR(tyParamOutDriver);
	fbFullMovAbsBl.tyParamInMove.diBacklashDistInUM	:= p_diMoveBacklashDistInUM;
	fbFullMovAbsBl.tyParamInMove.diAcc				:= p_diMoveAcc;
	fbFullMovAbsBl.tyParamInMove.diDec				:= p_diMoveDec;
	//fbFullMovAbsBl.tyParamInConvert					:= p_tyParamInConvert;
	fbFullMovAbsBl.bDir								:= p_bDir;
	fbFullMovAbsBl.bDirBl							:= p_bDirBl;
	fbFullMovAbsBl.bNoIndexPulse					:= p_bNoIndexPulse;
	fbFullMovAbsBl.eMotorType						:= p_eNtParamMotorType;
	fbFullMovAbsBl(bEn := FALSE);

	fbFullMovAbs.p_tyParamOutDriver					:= ADR(tyParamOutDriver);
	fbFullMovAbs.tyParamInMove.diBacklashDistInUM	:= p_diMoveBacklashDistInUM;
	fbFullMovAbs.tyParamInMove.diAcc				:= p_diMoveAcc;
	fbFullMovAbs.tyParamInMove.diDec				:= p_diMoveDec;
	fbFullMovAbs.tyParamInConvert					:= p_tyParamInConvert;
	fbFullMovAbs.bDir								:= p_bDir;
	fbFullMovAbs.bNoIndexPulse						:= p_bNoIndexPulse;
	fbFullMovAbs.eMotorType							:= p_eNtParamMotorType;
	fbFullMovAbs(bEn := FALSE);

	fbFullHm.p_tyParamOutDriver	:= ADR(tyParamOutDriver);
	fbFullHm.bDir				:= p_bDir;
	fbFullHm.bNoIndexPulse		:= p_bNoIndexPulse;
	fbFullHm.eMotorType			:= p_eNtParamMotorType;
	fbFullHm(bEn := FALSE);

	fbPwrOn.p_tyParamOutDriver	:= ADR(tyParamOutDriver);
	fbPwrOn.eMotorType			:= p_eNtParamMotorType;
	fbPwrOn(bEn := FALSE);

	fbPwrOff.p_tyParamOutDriver	:= ADR(tyParamOutDriver);
	fbPwrOff.eMotorType			:= p_eNtParamMotorType;
	fbPwrOff(bEn := FALSE);

	fbHoming.p_tyParamOutDriver	:= ADR(tyParamOutDriver);
	fbHoming.bDir				:= p_bDir;
	fbHoming.bNoIndexPulse		:= p_bNoIndexPulse;
	fbHoming.eMotorType			:= p_eNtParamMotorType;
	fbHoming(bEn := FALSE);

	fbMovAbs.p_tyParamOutDriver					:= ADR(tyParamOutDriver);
	fbMovAbs.tyParamInMove.diBacklashDistInUM	:= p_diMoveBacklashDistInUM;
	fbMovAbs.tyParamInMove.diAcc				:= p_diMoveAcc;
	fbMovAbs.tyParamInMove.diDec				:= p_diMoveDec;
	fbMovAbs.tyParamInConvert					:= p_tyParamInConvert;
	fbMovAbs.bDir								:= p_bDir;
	fbMovAbs.eMotorType							:= p_eNtParamMotorType;
	fbMovAbs(bEn := FALSE);

	fbMovRel.p_tyParamOutDriver					:= ADR(tyParamOutDriver);
	fbMovRel.tyParamInMove.diBacklashDistInUM	:= p_diMoveBacklashDistInUM;
	fbMovRel.tyParamInMove.diAcc				:= p_diMoveAcc;
	fbMovRel.tyParamInMove.diDec				:= p_diMoveDec;
	fbMovRel.tyParamInConvert					:= p_tyParamInConvert;
	fbMovRel.bDir								:= p_bDir;
	fbMovRel.eMotorType							:= p_eNtParamMotorType;
	fbMovRel(bEn := FALSE);

	fbJog.p_tyParamOutDriver	:= ADR(tyParamOutDriver);
	fbJog.tyParamInConvert		:= p_tyParamInConvert;
	fbJog.eMotorType			:= p_eNtParamMotorType;
	fbJog(bEn := FALSE);

	fbRstAxisErr.p_tyParamOutDriver	:= ADR(tyParamOutDriver);
	fbRstAxisErr(bEn := FALSE);

	fbStop.p_tyParamOutDriver	:= ADR(tyParamOutDriver);
	fbStop(bEn := FALSE);

	fbSDOWriteTorque.pDevice := ADR(p_sDevice);
	fbSDOWriteTorque.node	 := p_usiNode;
	fbSDOWriteTorque.index	 := 16#210C;
	fbSDOWriteTorque.subindex:= 0;
	fbSDOWriteTorque.datalen := 2;
	fbSDOWriteTorque(enable := FALSE);

	bModuleNotOK		:= TRUE;

END_ACTION
```

#### Act_InitLocal.st
```iecst
(** 2020-05-26 **)
ACTION Act_InitLocal:

	//Input Reference Link To Local Variable
	p_eAct ACCESS ADR(eAct);
	p_udiRstErr ACCESS ADR(udiRstErr);
	p_bPrep ACCESS ADR(bPrep);
	p_bEn ACCESS ADR(bEn);
	p_bDis ACCESS ADR(bDis);
	p_bOps ACCESS ADR(bOps);
	p_bManual ACCESS ADR(bManual);
	p_diWidthAtHmPos ACCESS ADR(diWidthAtHmPos);
	p_tyTuning ACCESS ADR(tyTuning);
	p_diGoWidth ACCESS ADR(diGoWidth);
	p_diJogVelInUMPS ACCESS ADR(diJogVelInUMPS);
	p_diMovePosInUM ACCESS ADR(diMovePosInUM);
	p_diMoveDistInUM ACCESS ADR(diMoveDistInUM);
	p_diMoveVelInUMPS ACCESS ADR(diMoveVelInUMPS);
	p_diMoveAcc ACCESS ADR(diMoveAcc);
	p_diMoveDec ACCESS ADR(diMoveDec);
	p_diMinAbsPosInUM ACCESS ADR(diMinAbsPosInUM);
	p_diMaxAbsPosInUM ACCESS ADR(diMaxAbsPosInUM);
	p_diMinWidthInUM ACCESS ADR(diMinWidthInUM);
	p_diMaxWidthInUM ACCESS ADR(diMaxWidthInUM);
	p_diWidthOffsetInUM ACCESS ADR(diWidthOffsetInUM);
	p_bInletSensor ACCESS ADR(bInletSensor);
	p_bOutletSensor ACCESS ADR(bOutletSensor);
	p_bClearSensor ACCESS ADR(bClearSensor);
	p_bMiddleSensor ACCESS ADR(bMiddleSensor);
	p_bInterruptSensor ACCESS ADR(bInterruptSensor);
	p_bOpenInterruptSensor ACCESS ADR(bOpenInterruptSensor);
	p_bCloseInterruptSensor ACCESS ADR(bCloseInterruptSensor);
	p_bDir ACCESS ADR(bDir);
	p_bDirBl ACCESS ADR(bDirBl);
	p_bNoIndexPulse ACCESS ADR(bNoIndexPulse);
	p_usiNode ACCESS ADR(usiNode);
	p_sDevice ACCESS ADR(sDevice);
	p_sProgNm ACCESS ADR(sProgNm);
	p_diMoveBacklashDistInUM ACCESS ADR(diMoveBacklashDistInUM);
	p_diPitchInUM ACCESS ADR(diPitchInUM);
	p_tyParamInHm ACCESS ADR(tyParamInHm);
	p_tyParamInConvert ACCESS ADR(tyParamInConvert);
	p_bNtSettingsLoadDone ACCESS ADR(bNtSettingsLoadDone);
	p_eNtParamMotorType ACCESS ADR(eMotorType);
	p_diServoTorque ACCESS ADR(diServoTorque);

END_ACTION
```

#### Act_Link.st
```iecst
(** 2019-03-29 **)
ACTION Act_Link:

//	IF p_bManual = TRUE THEN
//		p_diMoveVelInUMPS ACCESS p_UIMnlPPNomSpd;
//		p_diJogVelInUMPS ACCESS p_UIMnlPPJogSpd;
//	ELSE
//		p_diMoveVelInUMPS ACCESS p_NtParamAWAutoSpd;
//	END_IF

//	IF p_bProjInletShutPrep = TRUE THEN
//
//		IF p_bInletShutterCloseRS
//			THEN
//			bInterruptSensor1 := TRUE;
//		ELSE
//			bInterruptSensor1 := FALSE;
//		END_IF
//	ELSE
//		bInterruptSensor1 := FALSE;
//	END_IF

//	IF p_bProjOutletShutPrep = TRUE THEN
//		IF p_bOutletShutterCloseRS AND p_eAct = PPActJogOpen
//			THEN
//			bInterruptSensor2 := TRUE;
//		ELSE
//			bInterruptSensor2 := FALSE;
//		END_IF
//	ELSE
//		bInterruptSensor2 := FALSE;
//	END_IF

//	IF usiJogFwdStep = 40 AND p_eAct = PPActJogOpen THEN
//		p_bInterruptSensor	:= NOT p_bMagWidthChkSen;
//	END_IF
//
//	IF usiJogRevStep = 40 AND p_eAct = PPActJogClose THEN
//		p_bInterruptSensor  := NOT p_bMagWidthChkSen;
//	END_IF
//
//	IF p_eAct = PPActIdle OR p_eAct = PPActStop THEN
//		p_bInterruptSensor  := FALSE;
//	END_IF

//	p_bInterruptSensor := bInterruptSensor2 OR bInterruptSensor1;// OR p_bLinkSafetyRelay = FALSE;

END_ACTION
```

#### Act_LinkAction.st
```iecst
(** 2019-10-21 **)
ACTION Act_LinkAction:

//	IF eStatus = Idle THEN
		IF bModuleNotOK THEN
			p_eAct ACCESS ADR(eAct);
		ELSE
			IF p_bLinkStartupRun = TRUE THEN
				p_eAct ACCESS p_StartupServoPPAct;
			ELSIF p_bLinkOpsRun = TRUE OR p_bManual = TRUE THEN
				IF p_bLinkPullConvPullerExtCtrl AND NOT bJogFwdDone
					//AND NOT p_bLinkDIPullerExtRS
					THEN
						bJogStopDone := FALSE;

						CASE usiJogFwdStep OF

							0:

	//						diMtrPshrExtTrq    := 10 + (((p_diLinkProdRcpTrq -10)/10)*444/100);
							diMtrPshrExtTrq    := p_tyLinkTorqParam.usiStartTorque + (((p_diLinkProdRcpTrq -10)/10)*p_tyLinkTorqParam.uiRatio/100);

								IF p_bManual THEN
									memcpy(ADR(fbSDOWriteTorque.data0),p_UIMnlMtrPshrExtTorq,1);
									memcpy(ADR(fbSDOWriteTorque.data1),p_UIMnlMtrPshrExtTorq+1,1);
								ELSE
	//								memcpy(ADR(fbSDOWriteTorque.data0),p_ProdRcpCurrRcp1MtrPshrExtTorq,1);
	//								memcpy(ADR(fbSDOWriteTorque.data1),p_ProdRcpCurrRcp1MtrPshrExtTorq+1,1);

									memcpy(ADR(fbSDOWriteTorque.data0),ADR (diMtrPshrExtTrq),1);
									memcpy(ADR(fbSDOWriteTorque.data1),ADR(diMtrPshrExtTrq)+1,1);
								END_IF

								IF eStat <> PPActIdle THEN
									p_eAct := PPActIdle;
									usiJogFwdStep := 20;
								ELSE
									usiJogFwdStep := 20;
								END_IF

							20:
								fbSDOWriteTorque(enable := TRUE);
								IF fbSDOWriteTorque.status = 65535 THEN
									usiJogFwdStep := 22;
								END_IF

							22:
								fbSDOWriteTorque(enable := TRUE);
								IF fbSDOWriteTorque.status = 0 THEN
									fbSDOWriteTorque(enable := FALSE);
									usiJogFwdStep := 30;
								END_IF

							30:
								IF tyParamOut.bPwrOn = FALSE THEN
									p_eAct := PPActPwrOn;

									IF tyParamOut.bPwrOn THEN
										p_eAct := PPActIdle;
										usiJogFwdStep := 40;
									END_IF
								ELSE
									p_eAct := PPActIdle;
									usiJogFwdStep := 40;

								END_IF

						40:

								p_eAct := PPActJogOpen;

								IF EDGEPOS(p_bLinkDIPullerExtSlwRS) THEN
									p_eAct := PPActIdle;
								END_IF

							IF p_bLinkDIPullerExtSlwRS OR p_bLinkDIPullerExtRS  THEN

									p_diJogVelInUMPS := diExtSlowSpeed;

								ELSE
									IF p_bManual THEN
										p_diJogVelInUMPS ACCESS p_UIMnlPPJogSpd;
									ELSE
										p_diJogVelInUMPS := p_dintLinkPullerRetSpd * 3000;//290000/410000//51250//64062//Extend Speed
									END_IF
								END_IF

							//	IF (eStat = PPActJogOpen AND eMainStatus = Done)
							//		OR p_bLinkDIPullerExtRS
								IF p_bLinkDIPullerExtRS
									THEN
									p_eAct := PPActIdle;
	//								p_eAct := PPActStop;
									p_diJogVelInUMPS := 0;
									usiJogFwdStep := 50;

								END_IF

						50:
							p_eAct := PPActJogStop;
	//						p_eAct := PPActStop;
							p_diJogVelInUMPS := 0;
							IF (eStat = PPActJogStop AND eMainStatus = Done)
								THEN
								p_eAct := PPActIdle;
								usiJogFwdStep := 0;
								bJogFwdDone := TRUE;
							END_IF

						END_CASE

				ELSIF p_bLinkPullConvPullerRetCtrl AND NOT bJogRevDone
					//AND NOT p_bLinkDIPullerRetRS
					THEN

					bJogStopDone := FALSE;
					CASE usiJogRevStep OF

						0:
							memcpy(ADR(fbSDOWriteTorque.data0),ADR(udiMaxTorque),1);
							memcpy(ADR(fbSDOWriteTorque.data1),ADR(udiMaxTorque)+1,1);

							IF eStat <> PPActIdle THEN
								p_eAct := PPActIdle;
								usiJogRevStep := 20;
							ELSE
								usiJogRevStep := 20;
							END_IF

						20:
							fbSDOWriteTorque(enable := TRUE);
							IF fbSDOWriteTorque.status = 65535 THEN
								usiJogRevStep := 22;
							END_IF

						22:
							fbSDOWriteTorque(enable := TRUE);
							IF fbSDOWriteTorque.status = 0 THEN
								fbSDOWriteTorque(enable := FALSE);
								usiJogRevStep := 30;
							END_IF

						30:
							IF tyParamOut.bPwrOn = FALSE THEN
								p_eAct := PPActPwrOn;
								IF tyParamOut.bPwrOn THEN
									p_eAct := PPActIdle;
									usiJogRevStep := 40;
								END_IF
							ELSE
								p_eAct := PPActIdle;
								usiJogRevStep := 40;

							END_IF

						40:
							p_eAct := PPActJogClose;

							IF EDGEPOS(p_bLinkDIPullerRetSlwRS) THEN
								p_eAct := PPActIdle;
							END_IF

						IF p_bLinkDIPullerRetSlwRS OR p_bLinkDIPullerRetRS THEN

								p_diJogVelInUMPS := diSlowSpeed;
							ELSE
								IF p_bManual THEN
									p_diJogVelInUMPS ACCESS p_UIMnlPPJogSpd;
								ELSE
								p_diJogVelInUMPS :=  diRetSpd; //36250 //512500 //410000 //16000
								END_IF

							END_IF

						//	IF (eStat = PPActJogClose AND eMainStatus = Done)
						//		OR p_bLinkDIPullerRetRS
							IF p_bLinkDIPullerRetRS
								THEN
								p_eAct := PPActIdle;

								p_diJogVelInUMPS := 0;
								usiJogRevStep := 50;

							END_IF

						50:
							p_eAct := PPActJogStop;
							p_diJogVelInUMPS := 0;
							IF (eStat = PPActJogStop AND eMainStatus = Done)
							THEN
								p_eAct := PPActIdle;
								usiJogRevStep := 0;
								bJogRevDone := TRUE;
							END_IF

					END_CASE
				ELSE

					IF bJogStopDone = FALSE THEN
						p_eAct := PPActJogStop;
					END_IF

					usiJogFwdStep := 0;
					usiJogRevStep := 0;
					p_diJogVelInUMPS := 0;
					tyParamOutDriver.diJogVel_60FF := 0; // ADDED

					IF eStat = PPActJogStop AND eMainStatus = Done THEN
						p_eAct := PPActIdle;
						bJogStopDone := TRUE;
					END_IF

					IF tyParamInDriver.uiErrCode_603F <> 0 THEN //error 12592
						tyParamOutDriver.uiCtrlword_6040 := 0; //0111 (7)> 1111 (15)
					END_IF
				END_IF
			ELSE

				usiJogFwdStep := 0;
				usiJogRevStep := 0;
				p_diJogVelInUMPS := 0;
				IF eStatus <> Idle THEN
					p_eAct := PPActIdle;
					IF eStat = PPActIdle AND eMainStatus = Done THEN
						p_eAct := PPActIdle;
					END_IF
				END_IF
			END_IF
		END_IF
//	END_IF

	IF EDGENEG(p_bManual) OR EDGENEG(p_bLinkOpsRun) OR EDGENEG(p_bLinkStartupRun) THEN
		tyParamOutDriver.uiCtrlword_6040	:= 0;
	END_IF

	IF (eStat = PPActJogClose AND p_bLinkDIPullerRetRS)
		OR (eStat = PPActJogOpen AND p_bLinkDIPullerExtRS)
		THEN
		p_diJogVelInUMPS := 0;
	END_IF

	IF p_bLinkDIPullerRetRS = FALSE THEN
		bJogRevDone := FALSE;
	END_IF

	IF p_bLinkDIPullerExtRS = FALSE THEN
		bJogFwdDone := FALSE;
	END_IF
	//fbPwrOnDlyTmr
END_ACTION
```

#### Act_Main.st
```iecst
(** 2020-05-26 **)
ACTION Act_Main:

	//Main
IF bModuleNotOK = FALSE THEN

		CASE eStat OF

			PPActIdle:
				IF eStatus <> Idle THEN	//Reset Data
					//Private
					fbStop(bEn := FALSE);
					fbRstAxisErr(bEn := FALSE);
					fbJog(bEn := FALSE);
					fbMovRel(bEn := FALSE);
					fbMovAbs(bEn := FALSE);
					fbHoming(bEn := FALSE);
					fbPwrOff(bEn := FALSE);
					fbPwrOn(bEn := FALSE);
					fbFullHm(bEn := FALSE);
					fbFullMovAbs(bEn := FALSE);
					fbFullMovAbsBl(bEn := FALSE);
					fbSDOWrite(bEn := FALSE);
					fbTm(IN := FALSE);
					usiStep				:= 0;
					usiCount			:= 0;
					bNotInterruptible	:= FALSE;
					tyParamOutDriver.uiCtrlword_6040.7	:= FALSE;
					sStatTxt	:= a_sStatText[eStat];

				END_IF

				eStatus	:= Idle;

				IF EDGENEG(p_bManual) THEN
					fMotionCANRstCtrlWord(ADR(tyParamOutDriver));
				END_IF

			PPActGoWidth:
				IF (eStatus = Idle OR eStatus = Busy) THEN

					eStatus	:= Busy;

					sStatTxt	:= a_sStatText[eStat];

					bNotInterruptible	:= TRUE;

					CASE usiStep OF
						0:	//Wait For Motion Parameter Update
							p_diMovePosInUM	:= fAWWidthToPosInUM(p_diGoWidth , p_diWidthAtHmPos);
							usiStep	:= 1;

						1:	//Check Position Difference
							IF tyParamOut.bPosDiff = TRUE THEN
								usiStep	:= 2;
							ELSE
								eStatus	:= Done;
							END_IF

						2:	//Move
							fbFullMovAbsBl.tyParamInDriver					:= tyParamInDriver;
							fbFullMovAbsBl.tyParamInMove.diPosInUM			:= p_diMovePosInUM;
							fbFullMovAbsBl.tyParamInMove.diDistInUM			:= p_diMoveDistInUM;
							fbFullMovAbsBl.tyParamInMove.diVelInUMPS		:= p_diMoveVelInUMPS;
							fbFullMovAbsBl.tyParamInMove.diAcc				:= p_diMoveAcc;
							fbFullMovAbsBl.tyParamInMove.diDec				:= p_diMoveDec;
							fbFullMovAbsBl.tyParamOut						:= tyParamOut;
							fbFullMovAbsBl(bEn := TRUE);

							IF fbFullMovAbsBl.udiStatus = 0 THEN
								eStatus	:= Done;
							ELSIF fbFullMovAbsBl.udiStatus < 65534 THEN
								eStatus		:= Error;

								IF fbFullMovAbsBl.udiStatus = 1401 THEN
									udiStatus	:= 10002;	//Power On Time Out While Going New Width
								ELSIF fbFullMovAbsBl.udiStatus = 1402 THEN
									udiStatus	:= 10003;	//Homing Time Out While Going New Width
								ELSIF fbFullMovAbsBl.udiStatus = 1403 THEN
									udiStatus	:= 10004;	//Move Absolute Time Out While Going New Width
								ELSIF fbFullMovAbsBl.udiStatus = 1405 THEN
									udiStatus	:= 10005;	//Stop Motion Time Out While Going New Width
								ELSIF fbFullMovAbsBl.udiStatus = 1408 THEN
									udiStatus	:= 10006;	//Axis Error Reset Failed While Going New Width
								ELSIF fbFullMovAbsBl.udiStatus = 1409 THEN
									udiStatus	:= 10007;	//Axis Error Occur In Move Absolute While Going New Width
								ELSIF fbFullMovAbsBl.udiStatus = 1411 THEN
									udiStatus	:= 10008;	//Axis Error Occur In Homing While Going New Width
								ELSIF fbFullMovAbsBl.udiStatus = 1412 THEN
									udiStatus	:= 10009;	//Homing Done But Home Flag Is Not Activated While Going New Width
								ELSIF fbFullMovAbsBl.udiStatus = 1413 THEN
									udiStatus	:= 10010;	//Forward Limit Activated In Homing While Going New Width
								ELSIF fbFullMovAbsBl.udiStatus = 1414 THEN
									udiStatus	:= 10011;	//Reverse Limit Activated In Homing While Going New Width
								ELSIF fbFullMovAbsBl.udiStatus = 1415 THEN
									udiStatus	:= 10012;	//Forward Limit Activated In Move Absolute While Going New Width
								ELSIF fbFullMovAbsBl.udiStatus = 1416 THEN
									udiStatus	:= 10013;	//Reverse Limit Activated In Move Absolute While Going New Width
								ELSE
									udiStatus	:= fbFullMovAbsBl.udiStatus;
								END_IF
							END_IF

					END_CASE

				END_IF

			PPActGoWidthOff:
				IF (eStatus = Idle OR eStatus = Busy) THEN

					eStatus	:= Busy;

					sStatTxt	:= a_sStatText[eStat];

					bNotInterruptible	:= TRUE;

					CASE usiStep OF
						0:	//Wait For Motion Parameter Update
							p_diMovePosInUM	:= fAWWidthToPosInUM(p_diGoWidth , p_diWidthAtHmPos);
							usiStep	:= 1;

						1:	//Check Position Difference
							IF tyParamOut.bPosDiff = TRUE THEN
								usiStep	:= 2;
							ELSE
								eStatus	:= Done;
							END_IF

						2:	//Move
							fbFullMovAbsBl.tyParamInDriver					:= tyParamInDriver;
							fbFullMovAbsBl.tyParamInMove.diPosInUM			:= p_diMovePosInUM;
							fbFullMovAbsBl.tyParamInMove.diDistInUM			:= p_diMoveDistInUM;
							fbFullMovAbsBl.tyParamInMove.diVelInUMPS		:= p_diMoveVelInUMPS;
							fbFullMovAbsBl.tyParamInMove.diAcc				:= p_diMoveAcc;
							fbFullMovAbsBl.tyParamInMove.diDec				:= p_diMoveDec;
							fbFullMovAbsBl.tyParamOut						:= tyParamOut;
							fbFullMovAbsBl(bEn := TRUE);

							IF fbFullMovAbsBl.udiStatus = 0 THEN
								usiStep	:= 3;
							ELSIF fbFullMovAbsBl.udiStatus < 65534 THEN
								eStatus		:= Error;

								IF fbFullMovAbsBl.udiStatus = 1401 THEN
									udiStatus	:= 10035;	//Power On Time Out While Going New Width And Off
								ELSIF fbFullMovAbsBl.udiStatus = 1402 THEN
									udiStatus	:= 10036;	//Homing Time Out While Going New Width And Off
								ELSIF fbFullMovAbsBl.udiStatus = 1403 THEN
									udiStatus	:= 10037;	//Move Absolute Time Out While Going New Width And Off
								ELSIF fbFullMovAbsBl.udiStatus = 1405 THEN
									udiStatus	:= 10038;	//Stop Motion Time Out While Going New Width And Off
								ELSIF fbFullMovAbsBl.udiStatus = 1408 THEN
									udiStatus	:= 10039;	//Axis Error Reset Failed While Going New Width And Off
								ELSIF fbFullMovAbsBl.udiStatus = 1409 THEN
									udiStatus	:= 10040;	//Axis Error Occur In Move Absolute While Going New Width And Off
								ELSIF fbFullMovAbsBl.udiStatus = 1411 THEN
									udiStatus	:= 10041;	//Axis Error Occur In Homing While Going New Width And Off
								ELSIF fbFullMovAbsBl.udiStatus = 1412 THEN
									udiStatus	:= 10042;	//Homing Done But Home Flag Is Not Activated While Going New Width And Off
								ELSIF fbFullMovAbsBl.udiStatus = 1413 THEN
									udiStatus	:= 10043;	//Forward Limit Activated In Homing While Going New Width And Off
								ELSIF fbFullMovAbsBl.udiStatus = 1414 THEN
									udiStatus	:= 10044;	//Reverse Limit Activated In Homing While Going New Width And Off
								ELSIF fbFullMovAbsBl.udiStatus = 1415 THEN
									udiStatus	:= 10045;	//Forward Limit Activated In Move Absolute While Going New Width And Off
								ELSIF fbFullMovAbsBl.udiStatus = 1416 THEN
									udiStatus	:= 10046;	//Reverse Limit Activated In Move Absolute While Going New Width And Off
								ELSE
									udiStatus	:= fbFullMovAbsBl.udiStatus;
								END_IF
							END_IF

						3:	//Turn Off Motor
							fMotionCANRstCtrlWord(ADR(tyParamOutDriver));
							eStatus	:= Done;

					END_CASE

				END_IF

			PPActFullHm:
				IF (eStatus = Idle OR eStatus = Busy) THEN

					eStatus	:= Busy;

					sStatTxt	:= a_sStatText[eStat];

					bNotInterruptible	:= TRUE;

					fbFullHm.tyParamInDriver	:= tyParamInDriver;
					fbFullHm.tyParamOut			:= tyParamOut;
					fbFullHm(bEn := TRUE);

					IF fbFullHm.udiStatus = 0 THEN
						eStatus	:= Done;
					ELSIF fbFullHm.udiStatus < 65534 THEN
						eStatus		:= Error;

						IF fbFullHm.udiStatus = 1401 THEN
							udiStatus	:= 10014;	//Power On Time Out While Full Homing
						ELSIF fbFullHm.udiStatus = 1402 THEN
							udiStatus	:= 10015;	//Homing Time Out While Full Homing
						ELSIF fbFullHm.udiStatus = 1405 THEN
							udiStatus	:= 10016;	//Stop Motion Time Out While Full Homing
						ELSIF fbFullHm.udiStatus = 1408 THEN
							udiStatus	:= 10017;	//Axis Error Reset Failed While Full Homing
						ELSIF fbFullHm.udiStatus = 1411 THEN
							udiStatus	:= 10018;	//Axis Error Occur In Homing While Full Homing
						ELSIF fbFullHm.udiStatus = 1412 THEN
							udiStatus	:= 10019;	//Homing Done But Home Flag Is Not Activated While Full Homing
						ELSIF fbFullHm.udiStatus = 1413 THEN
							udiStatus	:= 10020;	//Forward Limit Activated In Homing While Full Homing
						ELSIF fbFullHm.udiStatus = 1414 THEN
							udiStatus	:= 10021;	//Reverse Limit Activated In Homing While Full Homing
						ELSE
							udiStatus	:= fbFullHm.udiStatus;
						END_IF
					END_IF

				END_IF

			PPActPwrOn:
				IF (eStatus = Idle OR eStatus = Busy) THEN

					eStatus	:= Busy;

					sStatTxt	:= a_sStatText[eStat];

					fbPwrOn.tyParamInDriver	:= tyParamInDriver;
					fbPwrOn(bEn := TRUE);

					IF fbPwrOn.udiStatus = 0 THEN
						eStatus	:= Done;
					ELSIF fbPwrOn.udiStatus < 65534 THEN
						eStatus		:= Error;

						IF fbPwrOn.udiStatus = 1401 THEN
							udiStatus	:= 10022;	//Power On Time Out
						ELSE
							udiStatus	:= fbPwrOn.udiStatus;
						END_IF
					END_IF

				END_IF

			PPActPwrOff:
				IF (eStatus = Idle OR eStatus = Busy) THEN

					eStatus	:= Busy;

					sStatTxt	:= a_sStatText[eStat];

					fbPwrOff.tyParamInDriver	:= tyParamInDriver;
					fbPwrOff(bEn := TRUE);

					IF fbPwrOff.udiStatus = 0 THEN
						eStatus	:= Done;
					ELSIF fbPwrOff.udiStatus < 65534 THEN
						eStatus		:= Error;

						IF fbPwrOff.udiStatus = 1400 THEN
							udiStatus	:= 10023;	//Power Off Time Out
						ELSE
							udiStatus	:= fbPwrOff.udiStatus;
						END_IF
					END_IF

				END_IF

			PPActHoming:

				IF (eStatus = Idle OR eStatus = Busy) THEN

					eStatus	:= Busy;

					sStatTxt	:= a_sStatText[eStat];

					bNotInterruptible	:= TRUE;

					fbHoming.tyParamInDriver	:= tyParamInDriver;
					fbHoming.tyParamOut			:= tyParamOut;
					fbHoming(bEn := TRUE);

					IF fbHoming.udiStatus = 0 THEN
						eStatus	:= Done;
					ELSIF fbHoming.udiStatus < 65534 THEN
						eStatus		:= Error;

						IF fbHoming.udiStatus = 1402 THEN
							udiStatus	:= 10024;	//Homing Time Out
						ELSIF fbHoming.udiStatus = 1411 THEN
							udiStatus	:= 10018;	//Axis Error Occur In Homing While Full Homing

						ELSIF fbHoming.udiStatus = 1413 THEN
							udiStatus	:= 10020;	//Forward Limit Activated In Homing While Full Homing
						ELSIF fbHoming.udiStatus = 1414 THEN
							udiStatus	:= 10021;	//Reverse Limit Activated In Homing While Full Homing
						ELSE
							udiStatus	:= fbHoming.udiStatus;
						END_IF
					END_IF

				END_IF

			PPActMovAbs:
				IF (eStatus = Idle OR eStatus = Busy) THEN

					eStatus	:= Busy;

					sStatTxt	:= a_sStatText[eStat];

					bNotInterruptible	:= TRUE;

					fbMovAbs.tyParamInDriver			:= tyParamInDriver;
					fbMovAbs.tyParamInMove.diPosInUM	:= p_diMovePosInUM;
					fbMovAbs.tyParamInMove.diDistInUM	:= p_diMoveDistInUM;
					fbMovAbs.tyParamInMove.diVelInUMPS	:= p_diMoveVelInUMPS;
					fbMovAbs.tyParamInMove.diAcc		:= p_diMoveAcc;
					fbMovAbs.tyParamInMove.diDec		:= p_diMoveDec;
					fbMovAbs(bEn := TRUE);

					IF fbMovAbs.udiStatus = 0 THEN
						eStatus	:= Done;
					ELSIF fbMovAbs.udiStatus < 65534 THEN
						eStatus		:= Error;

						IF fbMovAbs.udiStatus = 1403 THEN
							udiStatus	:= 10025;	//Move Absolute Time Out
						ELSE
							udiStatus	:= fbMovAbs.udiStatus;
						END_IF
					END_IF

				END_IF

			PPActMovRel:
				IF (eStatus = Idle OR eStatus = Busy) THEN

					eStatus	:= Busy;

					sStatTxt	:= a_sStatText[eStat];

					bNotInterruptible	:= TRUE;

					fbMovRel.tyParamInDriver			:= tyParamInDriver;
					fbMovRel.tyParamInMove.diPosInUM	:= p_diMovePosInUM;
					fbMovRel.tyParamInMove.diDistInUM	:= p_diMoveDistInUM;
					fbMovRel.tyParamInMove.diVelInUMPS	:= p_diMoveVelInUMPS;
					fbMovRel.tyParamInMove.diAcc		:= p_diMoveAcc;
					fbMovRel.tyParamInMove.diDec		:= p_diMoveDec;
					fbMovRel(bEn := TRUE);

					IF fbMovRel.udiStatus = 0 THEN
						eStatus	:= Done;
					ELSIF fbMovRel.udiStatus < 65534 THEN
						eStatus		:= Error;

						IF fbMovRel.udiStatus = 1404 THEN
							udiStatus	:= 10026;	//Move Relative Time Out
						ELSE
							udiStatus	:= fbMovRel.udiStatus;
						END_IF
					END_IF

				END_IF

			PPActJogOpen:
				IF (eStatus = Idle OR eStatus = Busy) THEN

					eStatus	:= Busy;

					sStatTxt	:= a_sStatText[eStat];

					bNotInterruptible	:= TRUE;

					fbJog.tyParamInDriver	:= tyParamInDriver;
					fbJog.tyParamInMove.diAcc		:= p_diMoveAcc;
					fbJog.tyParamInMove.diDec		:= p_diMoveDec;

					IF p_bDir = TRUE THEN
						fbJog.tyParamInJog.diVelInUMPS	:= p_diJogVelInUMPS;
					ELSE
						fbJog.tyParamInJog.diVelInUMPS	:= p_diJogVelInUMPS * -1;
					END_IF

					fbJog(bEn := TRUE);

					IF fbJog.udiStatus = 0 THEN
						bJogging	:= TRUE;
						bJogOpen	:= TRUE;
						eStatus		:= Done;
					ELSIF fbJog.udiStatus < 65534 THEN
						udiStatus	:= fbJog.udiStatus;
						eStatus		:= Error;
					END_IF

				END_IF

			PPActJogClose:
				IF (eStatus = Idle OR eStatus = Busy) THEN

					eStatus	:= Busy;

					sStatTxt	:= a_sStatText[eStat];

					bNotInterruptible	:= TRUE;

					fbJog.tyParamInDriver			:= tyParamInDriver;
					fbJog.tyParamInMove.diAcc		:= p_diMoveAcc;
					fbJog.tyParamInMove.diDec		:= p_diMoveDec;

					IF p_bDir = TRUE THEN
						fbJog.tyParamInJog.diVelInUMPS	:= p_diJogVelInUMPS * -1;
					ELSE
						fbJog.tyParamInJog.diVelInUMPS	:= p_diJogVelInUMPS;
					END_IF

					fbJog(bEn := TRUE);

					IF fbJog.udiStatus = 0 THEN
						bJogging	:= TRUE;
						bJogClose	:= TRUE;
						eStatus		:= Done;
					ELSIF fbJog.udiStatus < 65534 THEN
						udiStatus	:= fbJog.udiStatus;
						eStatus		:= Error;
					END_IF

				END_IF

			PPActJogStop:
				IF (eStatus = Idle OR eStatus = Busy) THEN

					sStatTxt	:= a_sStatText[eStat];

					fMotionCANJogStop(ADR(tyParamOutDriver));
					bJogging	:= FALSE;
					bJogClose	:= FALSE;
					bJogOpen	:= FALSE;
					eStatus	:= Done;

				END_IF

			PPActRstAxisErr:
				IF (eStatus = Idle OR eStatus = Busy) THEN

					eStatus	:= Busy;

					sStatTxt	:= a_sStatText[eStat];

					fbRstAxisErr(bEn := TRUE);

					IF fbRstAxisErr.udiStatus = 0 THEN
						eStatus	:= Done;
					ELSIF fbRstAxisErr.udiStatus < 65534 THEN
						udiStatus	:= fbRstAxisErr.udiStatus;
						eStatus		:= Error;
					END_IF

				END_IF

			PPActStop:
				IF (eStatus = Idle OR eStatus = Busy) THEN

					eStatus	:= Busy;

					sStatTxt	:= a_sStatText[eStat];

					fbStop.tyParamInDriver	:= tyParamInDriver;
					fbStop(bEn := TRUE);

					IF fbStop.udiStatus = 0 THEN
						bJogging	:= FALSE;
						bJogClose	:= FALSE;
						bJogOpen	:= FALSE;
						eStatus		:= Done;
					ELSIF fbStop.udiStatus < 65534 THEN
						eStatus		:= Error;

						IF fbStop.udiStatus = 1405 THEN
							udiStatus	:= 10027;	//Stop Motion Time Out
						ELSE
							udiStatus	:= fbStop.udiStatus;
						END_IF
					END_IF

				END_IF

			PPActSDOWrite:
				IF (eStatus = Idle OR eStatus = Busy) THEN

					eStatus	:= Busy;

					sStatTxt	:= a_sStatText[eStat];

					fbTm(IN := TRUE);

					IF fbTm.Q THEN

						fbSDOWrite.tyParamOut	:= tyParamOut;
						fbSDOWrite.tyTuning.diAsdaA2AntiInterGain	:= p_tyTuning.diAsdaA2AntiInterGain;
						fbSDOWrite.tyTuning.diAsdaA2Inertia			:= p_tyTuning.diAsdaA2Inertia;
						fbSDOWrite.tyTuning.diAsdaA2LowPassFltr		:= p_tyTuning.diAsdaA2LowPassFltr;
						fbSDOWrite.tyTuning.diAsdaA2PosFFGain		:= p_tyTuning.diAsdaA2PosFFGain;
						fbSDOWrite.tyTuning.diAsdaA2PosLoopGain		:= p_tyTuning.diAsdaA2PosLoopGain;
						fbSDOWrite.tyTuning.diAsdaA2SpdIntegral		:= p_tyTuning.diAsdaA2SpdIntegral;
						fbSDOWrite.tyTuning.diAsdaA2SpdLoopGain		:= p_tyTuning.diAsdaA2SpdLoopGain;
						fbSDOWrite.tyTuning.diAsdaA2FirstTorqueCmd	:= p_diServoTorque;

						fbSDOWrite(bEn := TRUE);

						IF fbSDOWrite.udiStatus = 0 THEN
							eStatus	:= Done;
						ELSIF fbSDOWrite.udiStatus < 65534 THEN
							fMotionCANRstCtrlWord(ADR(tyParamOutDriver));

							IF usiCount < 5 THEN
								fbTm(IN := FALSE);
								fbSDOWrite(bEn := FALSE);

								usiCount	:= usiCount + 1;
							ELSE
								eStatus	:= Error;

								IF fbSDOWrite.udiStatus = 1406 THEN
									udiStatus	:= 10028;	//SDO Write Error
								ELSE
									udiStatus	:= fbSDOWrite.udiStatus;
								END_IF
							END_IF

						END_IF

					END_IF

				END_IF
		END_CASE

ELSE
	CASE eStat OF
		PPActSDOWrite:
			IF (eStatus = Idle OR eStatus = Busy) THEN

				eStatus	:= Busy;

				sStatTxt	:= a_sStatText[eStat];

				fbTm(IN := TRUE);

				IF fbTm.Q THEN

					fbSDOWrite.tyParamOut	:= tyParamOut;
					fbSDOWrite.tyTuning		:= p_tyTuning;

					fbSDOWrite(bEn := TRUE);

					IF fbSDOWrite.udiStatus = 0 THEN
						eStatus	:= Done;
					ELSIF fbSDOWrite.udiStatus < 65534 THEN
						fMotionCANRstCtrlWord(ADR(tyParamOutDriver));

						IF usiCount < 5 THEN
							fbTm(IN := FALSE);
							fbSDOWrite(bEn := FALSE);

							usiCount	:= usiCount + 1;
						ELSE
							eStatus	:= Error;

							IF fbSDOWrite.udiStatus = 1406 THEN
								udiStatus	:= 10028;	//SDO Write Error
							ELSE
								udiStatus	:= fbSDOWrite.udiStatus;
							END_IF
						END_IF

					END_IF

				END_IF

			END_IF

		PPActBGStartModOKChk:
			IF (eStatus = Idle OR eStatus = Busy) THEN

				sStatTxt	:= a_sStatText[eStat];

				bModuleOKChk	:= TRUE;
				eStatus			:= Done;

			END_IF

		PPActBGStopModOKChk:
			IF (eStatus = Idle OR eStatus = Busy) THEN

				sStatTxt	:= a_sStatText[eStat];

				bModuleOKChk	:= FALSE;
				eStatus			:= Done;

			END_IF

		PPActIdle:
			IF eStatus <> Idle THEN	//Reset Data
				//Private
				fbStop(bEn := FALSE);
				fbRstAxisErr(bEn := FALSE);
				fbJog(bEn := FALSE);
				fbMovRel(bEn := FALSE);
				fbMovAbs(bEn := FALSE);
				fbHoming(bEn := FALSE);
				fbPwrOff(bEn := FALSE);
				fbPwrOn(bEn := FALSE);
				fbFullHm(bEn := FALSE);
				fbFullMovAbs(bEn := FALSE);
				fbFullMovAbsBl(bEn := FALSE);
				fbSDOWrite(bEn := FALSE);
				fbTm(IN := FALSE);
				usiStep				:= 0;
				usiCount			:= 0;
				bNotInterruptible	:= FALSE;
				tyParamOutDriver.uiCtrlword_6040.7	:= FALSE;

				sStatTxt	:= a_sStatText[eStat];

			END_IF

			eStatus	:= Idle;

			IF EDGENEG(p_bManual) THEN
				fMotionCANRstCtrlWord(ADR(tyParamOutDriver));
			END_IF

		PPActRstNode:
			IF (eStatus = Idle OR eStatus = Busy) THEN

				eStatus	:= Busy;

				sStatTxt	:= a_sStatText[eStat];
				IF bRstErr THEN
					fbModuleOK(bEn := FALSE, bModuleOK := bModuleOK);
				END_IF
				fbModuleOK(bEn := TRUE);
				IF fbModuleOK.udiStatus = 0 THEN
					fbModuleOK(bEn := FALSE);
					eStatus			:= Done;
				ELSIF fbModuleOK.udiStatus < 65534 THEN
					eStatus		:= Error;

					IF fbModuleOK.udiStatus = 1407 THEN
						udiStatus	:= 10001;	//CANOpen Communication Error, ModuleOK Not TRUE
						fbModuleOK(bEn := FALSE);
					ELSE
						udiStatus	:= fbModuleOK.udiStatus;
					END_IF
				END_IF
			END_IF

		PPActRstAxisErr:
			IF (eStatus = Idle OR eStatus = Busy) THEN

				eStatus	:= Busy;

				sStatTxt	:= a_sStatText[eStat];

				fbRstAxisErr(bEn := TRUE);

				IF fbRstAxisErr.udiStatus = 0 THEN
					eStatus	:= Done;
				ELSIF fbRstAxisErr.udiStatus < 65534 THEN
					udiStatus	:= fbRstAxisErr.udiStatus;
					eStatus		:= Error;
				END_IF

			END_IF

	END_CASE
END_IF

END_ACTION
```

#### Act_RstErr.st
```iecst
(** 2020-03-16 **)
ACTION Act_RstErr:

	IF p_udiRstErr <> udiRstErrOld THEN
		bRstErr			:= TRUE;
		udiRstErrOld	:= p_udiRstErr;
		tyParamOutDriver.diJogVel_60FF := 0;
	ELSE
		bRstErr			:= FALSE;
	END_IF

	tyParamOutDriver.uiCtrlword_6040.7	:= bRstErr;

END_ACTION
```

#### Cyclic.st
```iecst
(** 2020-03-16 **)
PROGRAM _CYCLIC

	IF bInitDone = FALSE THEN
		bInitDone	:= TRUE;

		Act_InitLocal;
		Act_InitGlobal;

	ELSIF bInitialDone = FALSE THEN
		IF p_bNtSettingsLoadDone = TRUE THEN
			bInitialDone	:= TRUE;

			Act_Initial;
		END_IF

	ELSE

		Act_RstErr;
		Act_LinkAction;
		Act_Action;
		Act_LinkEn;

		IF EDGEPOS(p_bDis = FALSE) THEN
			bModuleNotOK := TRUE;
		END_IF

		IF (p_bPrep = TRUE) AND (p_bEn = TRUE) AND (p_bDis = FALSE) THEN
			Act_Link;
			Act_Background;
			Act_Main;
		ELSE
			Act_Main_Disable;

			IF eStat <> PPActIdle THEN
				eStatus	:= Done;
			ELSE
				eStatus	:= Idle;
			END_IF
		END_IF

		Act_CombineErr;
		Act_Alarm;
		Act_Alarm1;
		Act_Alarm2;
		Act_Alarm3;

	END_IF

END_PROGRAM
```

#### Init.st
```iecst
(** 2019-04-24 **)
PROGRAM _INIT

	(* Always Change If Project Change *)

	//Pass Address To Global Address For External Use
	//Action, State & Status
	p_PPStat	:= ADR(eStat);
	p_PPStatus	:= ADR(eMainStatus);
	p_PPStatTxt	:= ADR(sStatTxt);

	//Alarm
	p_PPAlmData		:= ADR(tyAlmData);
	p_PPAlmData1	:= ADR(tyAlmData1);
	p_PPAlmData2	:= ADR(tyAlmData2);
	p_PPAlmData3	:= ADR(tyAlmData3);

	//Output
	p_PPParamOut		:= ADR(tyParamOut);
	p_PPPwrOn			:= ADR(tyParamOut.bPwrOn);
	p_PPIsHomed			:= ADR(tyParamOut.bIsHomed);
	p_PPPosDiff			:= ADR(tyParamOut.bPosDiff);
	p_PPAxisErr			:= ADR(tyParamOut.bAxisErr);
	p_PPAxisErrID		:= ADR(tyParamOut.udiAxisErrID);
	p_PPFwdLmtSen		:= ADR(tyParamOut.bFwdLmtSen);
	p_PPRevLmtSen		:= ADR(tyParamOut.bRevLmtSen);
	p_PPActualPos		:= ADR(tyParamOut.diActualPosInUM);
	p_PPAxisErrTxt		:= ADR(sAxisErrTxt);
	p_PPWidthPosDiff	:= ADR(bWidthPosDiff);
	p_PPJogging			:= ADR(bJogging);
	p_PPExtSen			:= ADR(bOpenSen);
	p_PPRetSen			:= ADR(bCloseSen);

	(* Always Change If Project Change *)

END_PROGRAM
```

### Readme.txt
```
Program
TCP - AGVTCP
TCPTop - Scanner scan on top
TCPBtm - Scanner scan on bottom.
```

### TCP.typ - Do Not Change!!!
```iecst
(*2019-05-04*)
(**)
(*Action*)

TYPE
	eTCPAction :
		(
		TCPActIdle,
		TCPActCreateDir,
		TCPActDeleteOldLog
		);
END_TYPE

(**)

TYPE
	tyTCPHistoryMsg : 	STRUCT
		eTCP : eTCPMsgType;
		sMsg : STRING[200];
	END_STRUCT;
	eTCPMsgType :
		(
		MsgNA,
		MsgRcvFromTCP,
		MsgSndToTCP
		);
	tyAIVMsgRcvDat : 	STRUCT
		bEnterPW : BOOL;
		bELD1Reached : BOOL;
		bELD1Completed : BOOL;
		bELD2Reached : BOOL;
		bELD2Completed : BOOL;
		bELD3Reached : BOOL;
		bELD3Completed : BOOL;
		bEUL1Reached : BOOL;
		bEUL1Completed : BOOL;
		bEUL2Reached : BOOL;
		bEUL2Completed : BOOL;
		bEUL3Reached : BOOL;
		bEUL3Completed : BOOL;
		bStandbyReached : BOOL;
		bStandbyCompleted : BOOL;
		bLocalizeCompleted : BOOL;
		bMoveBackCompleted : BOOL;
		bLoginSuccess : BOOL;
		bOneLineStatus : BOOL;
	END_STRUCT;
END_TYPE

(**)
(**)
(*Server Action*)

TYPE
	eTCPSvrAction :
		(
		SvrActIdle,
		SvrActRead,
		SvrActRead1,
		SvrActWrite
		);
	eTCPClientServer :
		(
		Client,
		Server
		);
	eTCPAGVStatus :
		(
		AGVNA := 10,
		AGVError := 11,
		AGVReady := 12,
		AGVAvailable := 13,
		AGV2NA := 20,
		AGV2Error := 21,
		AGV2Ready := 22,
		AGV2Available := 23,
		AGV3NA := 30,
		AGV3Error := 31,
		AGV3Ready := 32,
		AGV3Available := 33,
		AGV4NA := 40,
		AGV4Error := 41,
		AGV4Ready := 42,
		AGV4Available := 43
		);
	tyTCPAGVDetail : 	STRUCT
		sAGVMag : STRING[10];
		eAGVStatus : eTCPAGVStatus;
		usiAGVReq : USINT; (*0: To Bring, 1:To Get*)
	END_STRUCT;
END_TYPE

(**)
(*Scanner Action*)

TYPE
	eTCPAction1 :
		(
		TCPActIdle_0,
		TCPActFullWriteRead,
		TCPActFullWriteReadUntilValid,
		TCPActDebug
		);
END_TYPE

(**)

TYPE
	tyTCP : 	STRUCT
		In : tyTCPIn1;
		Out : tyTCPOut1;
	END_STRUCT;
	tyTCPIn1 : 	STRUCT
		bManual : BOOL;
		eAct : eTCPAction;
		udiRstErr : UDINT;
		bPrep : BOOL;
		bEn : BOOL;
		bDis : BOOL;
		sSvrIP : STRING[15];
		uiSvrPort : UINT;
		uiClientPort : UINT;
		sMsgSnd : STRING[65535];
		sIPAddr : STRING[15];
		tyDTStructure : DTStructure;
		dtCurrDT : DATE_AND_TIME;
		eTCPModel : eTCPClientServer;
		bFltrIP : BOOL;
		bFltrPort : BOOL;
		sAllwClntIP : STRING[15];
		uiAllwClntPort : UINT;
		bReconnect : BOOL;
		udiSndBffrSize : UDINT;
		udiRcvBffrSize : UDINT;
		udiAliveIdleTimeInSec : UDINT;
		tConnTimeOut : TIME;
		bOpsRun : BOOL;
		usiProjMag : USINT;
		sProgNm : STRING[15];
		bNtSettingsLoadDone : BOOL;
		udiFileKeepDay : UDINT;
		tyDTMagToAGV : tyTagDTMagToAGV;
		bUSB : BOOL;
		bUSB2 : BOOL;
		bDBA : BOOL;
		bDBA2 : BOOL;
		bLinkStartupRun : BOOL;
		bLinkUIClearMsg : BOOL;
		bLinkConnectEn : BOOL;
		eLinkAGVComProtocol : eMcAGVCommProtocol;
	END_STRUCT;
	tyTCPOut1 : 	STRUCT
		eStat : eMagConv2ClpAction;
		eStatus : eFBStatus;
		sStatTxt : STRING[200];
		tyAlmData : tyAlmDat;
		tyAlmData1 : tyAlmDat;
		tyAlmData2 : tyAlmDat;
		tyAlmData3 : tyAlmDat;
		bConnected : BOOL;
		sExtractBatteryLvl : USINT;
		rCurrentBatteryLvl : USINT;
		bUBA : BOOL;
		bUBA2 : BOOL;
		bDSB : BOOL;
		bDSB2 : BOOL;
		tyAIVMsgRcvData : tyAIVMsgRcvDat;
		sSvrMsgRcv : STRING[65535];
		eMagAGVStatus : ARRAY[0..7]OF eTCPAGVStatus;
	END_STRUCT;
END_TYPE
```

### TCP.var - Change By Project
```iecst
(*2020-09-10*)
(**)
(*Action & State & Status*)
VAR
	p_TCPStat : UDINT;
	p_TCPStatus : UDINT;
	p_TCPStatTxt : UDINT;
END_VAR
(**)
(*Alarm*)
VAR
	p_TCPAlmData : UDINT;
	p_TCPAlmData1 : UDINT;
	p_TCPAlmData2 : UDINT;
	p_TCPAlmData3 : UDINT;
END_VAR
(**)
(*Output*)
VAR
	p_TCPAIVBatteryLvl : UDINT;
	p_TCPAIVCurrentBatteryLvl : UDINT;
	p_TCPConnected : UDINT;
	p_TCPHistoryList : UDINT;
	p_TCPMsgRcvData : UDINT;
	p_TCPSvrMsgRcvData : UDINT;
	p_TCPSvrAGVStatus1 : UDINT;
	p_TCPSvrAGVStatus2 : UDINT;
	p_TCPSvrAGVStatus3 : UDINT;
	p_TCPSvrAGVStatus4 : UDINT;
END_VAR
(**)
VAR
	p_TCPSvrUBA : UDINT;
	p_TCPSvrUBA2 : UDINT;
	p_TCPSvrDSB : UDINT;
	p_TCPSvrDSB2 : UDINT;
END_VAR
```

### Program Logical/TCP/TCP (IEC, version 1.00.0) - 1.00.0 - NtHermes v5.00.0 , NtTCP v5.00.0 , NtMessage v5.00.0

#### Act_InputConfig.st - Change By Project
```iecst
(** 2019-06-28 **)
ACTION Act_InputConfig:

	(* Always Change If Project Change *)

	//Pass Data To Link
//	p_bLinkStartupRun ACCESS p_StartupRun;
//	p_bLinkUIClearMsg ACCESS p_UITCPClearMsg;
//	p_bLinkConnectEn ACCESS p_UITCPConnectionEn;
	p_bUSB ACCESS p_USSOT1USB;
	p_bUSB2 ACCESS p_USSOT2USB;
	p_bDBA ACCESS p_DSSOT1DBA;
	p_bDBA2 ACCESS p_DSSOT2DBA;
	p_eLinkAGVComProtocol ACCESS p_McParamAGVComProtocol;

	//Pass Data To Internal Use
	//	p_bManual ACCESS p_UIUIMnlMod;
	p_udiRstErr ACCESS p_RstErrReset;
	p_sIPAddr ACCESS p_HWInfoIPAddr;
	p_tyDTStructure ACCESS p_TimeCurrDTStruct;
	p_dtCurrDT ACCESS p_TimeCurrDT;
	p_bOpsRun ACCESS p_OpsRun;
	p_sMsgSnd ACCESS ADR(sMsgSnd);
	p_sSvrIP ACCESS p_HWInfoIPAddr;
	p_uiSvrPort ACCESS p_McParamTCPSvrPort; //UI setting input

	p_usiProjMag ACCESS p_NtParamProjMag;

	p_bNtSettingsLoadDone ACCESS p_StartupNtSettingsLoadDone;

	(* Always Change If Project Change *)

	//Link bPrep, bEn & bDis
	bEn := p_eLinkAGVComProtocol = McSetAGVTCPEnableTCP;

	IF p_bEn THEN
		bRun := TRUE;
	ELSE
		bRun := FALSE;
	END_IF

END_ACTION
```

#### Act_OutputConfig.st - Change By Project
```iecst
(** 2020-09-10 **)
PROGRAM _INIT

	(* Always Change If Project Change *)

	//Pass Address To Global Address For External Use
	//Action, State & Status
	p_TCPStat		:= ADR(eStat);
	p_TCPStatus		:= ADR(eMainStatus);
	p_TCPStatTxt	:= ADR(sStatTxt);

	//Alarm
	p_TCPAlmData	:= ADR(tyAlmData);
	p_TCPAlmData1	:= ADR(tyAlmData1);
	p_TCPAlmData2	:= ADR(tyAlmData2);
	p_TCPAlmData3	:= ADR(tyAlmData3);

	//Output
	p_TCPConnected				:= ADR(bConnected);
	p_TCPHistoryList			:= ADR(a_tyHistoryList);
	p_TCPAIVBatteryLvl			:= ADR(sExtractBatteryLvl);
	p_TCPAIVCurrentBatteryLvl	:= ADR(rCurrentBatteryLvl);
	p_TCPMsgRcvData				:= ADR(tyAIVMsgRcvData); //Client

	p_TCPSvrMsgRcvData			:= ADR(sSvrMsgRcv);
	p_TCPSvrAGVStatus1			:= ADR(eMagAGVStatus[0]);
	p_TCPSvrAGVStatus2			:= ADR(eMagAGVStatus[1]);
	p_TCPSvrAGVStatus3			:= ADR(eMagAGVStatus[2]);
	p_TCPSvrAGVStatus4			:= ADR(eMagAGVStatus[3]);

	p_TCPSvrUBA					:= ADR(bUBA);
	p_TCPSvrUBA2				:= ADR(bUBA2);
	p_TCPSvrDSB					:= ADR(bDSB);
	p_TCPSvrDSB2				:= ADR(bDSB2);
	(* Always Change If Project Change *)

END_PROGRAM
ACTION Act_OutputConfig:

	g_tyTCP := tylocalTCP.Out; // Change the Global Naming According to the Physical Hardware Module

END_ACTION
```

#### InputRef_Link.var - Change By Project
```iecst
(*2019-06-28*)
(**)
VAR
	p_bLinkStartupRun : REFERENCE TO BOOL;
	p_bLinkUIClearMsg : REFERENCE TO BOOL;
	p_bLinkConnectEn : REFERENCE TO BOOL;
	p_eLinkAGVComProtocol : REFERENCE TO eMcAGVCommProtocol;
END_VAR
```

#### Act_LinkAction.st - Change By Project
```iecst
(** 2019-04-09 **)
ACTION Act_LinkAction:

//	IF p_bLinkStartupRun = TRUE THEN
//		p_eAct ACCESS p_StartupTCPAct;
//	ELSE
//		p_eAct ACCESS ADR(eAct);
//
//		IF p_bManual THEN
//			IF EDGEPOS(p_bLinkConnectEn) THEN
//				bRun	:= TRUE;
//				bStop	:= FALSE;
//			END_IF
//
//			IF EDGENEG(p_bLinkConnectEn) THEN
//				bStop	:= TRUE;
//			END_IF
//		ELSE
//			bRun	:= TRUE;
//			bStop	:= FALSE;
//		END_IF
//
//
//	END_IF

END_ACTION
```

#### Act_LinkEn.st - Change By Project
```iecst
(** 2019-03-15 **)
ACTION Act_LinkEn:

END_ACTION
```

#### Act_Link.st - Change By Project
```iecst
(** 2019-06-04 **)
ACTION Act_Link:

//	IF p_bManual THEN
//		p_sMsgSnd ACCESS p_UITCPAIVSndMsg;
//	ELSE
//		p_sMsgSnd ACCESS p_OpsTCPAIVSndMsg;
//	END_IF

END_ACTION
```

#### Cyclic.st - Do Not Change!!!
```iecst
(** 2020-09-10 **)
PROGRAM _CYCLIC

	IF bInitDone = FALSE THEN
		bInitDone	:= TRUE;

		Act_InitLocal;
		Act_InitGlobal;

	ELSIF bInitialDone = FALSE THEN
		IF p_bNtSettingsLoadDone = TRUE THEN
			bInitialDone	:= TRUE;

			Act_Initial;
		END_IF

	ELSE

		Act_RstErr;
		Act_LinkAction;
		Act_Action;
		Act_LinkEn;

		IF (p_bPrep = TRUE) AND (p_bEn = TRUE) AND (p_bDis = FALSE) THEN
			Act_Link;
			Act_Main;
			Act_Background;

		ELSE
			Act_Main_Disable;

			IF eStat <> TCPActIdle THEN
				eStatus	:= Done;
			ELSE
				eStatus	:= Idle;
			END_IF

		END_IF

		Act_Alarm;

	END_IF

END_PROGRAM
```

#### Act_InitLocal.st - Do Not Change!!!
```iecst
(** 2019-06-28 **)
ACTION Act_InitLocal:

	//Input Reference Link To Local Variable
	p_eAct ACCESS ADR(eAct);
	p_udiRstErr ACCESS ADR(udiRstErr);
	p_bPrep ACCESS ADR(bPrep);
	p_bEn ACCESS ADR(bEn);
	p_bDis ACCESS ADR(bDis);
	p_bManual ACCESS ADR(bManual);
	p_sIPAddr ACCESS ADR(sIPAddr);
	p_tyDTStructure ACCESS ADR(tyDTStructure);
	p_dtCurrDT ACCESS ADR(dtCurrDT);
	p_udiSndBffrSize ACCESS ADR(udiSndBffrSize);
	p_udiRcvBffrSize ACCESS ADR(udiRcvBffrSize);
	p_udiAliveIdleTimeInSec ACCESS ADR(udiAliveIdleTimeInSec);
	p_tConnTimeOut ACCESS ADR(tConnTimeOut);
	p_bOpsRun ACCESS ADR(bOpsRun);
	p_udiFileKeepDay ACCESS ADR(udiFileKeepDay);
	p_sProgNm ACCESS ADR(sProgNm);
	p_bNtSettingsLoadDone ACCESS ADR(bNtSettingsLoadDone);
	p_sMsgSnd ACCESS ADR(sMsgSnd);
	p_sSvrIP ACCESS ADR(sSvrIP);
	p_uiSvrPort ACCESS ADR(uiSvrPort);
	p_uiClientPort ACCESS ADR(uiClientPort);

	p_eTCPModel ACCESS ADR (eTCPModel);
	p_bFltrIP ACCESS ADR(bFltrIP);
	p_bFltrPort ACCESS ADR(bFltrPort);
	p_sAllwClntIP ACCESS ADR(sAllwClntIP);
	p_uiAllwClntPort ACCESS ADR(uiAllwClntPort);
	p_bReconnect ACCESS ADR(bReconnect);

	p_usiProjMag ACCESS ADR(usiProjMag);
	p_bUSB ACCESS ADR(bUSB);
	p_bUSB2 ACCESS ADR(bUSB2);
	p_bDBA ACCESS ADR(bDBA);
	p_bDBA2 ACCESS ADR(bDBA2);

	//Machine status
	p_tyDTMagToAGV ACCESS ADR(tyDTMagToAGV);
//	p_tyDTMagToAGV1 ACCESS ADR(tyDTMagToAGV1);
//	p_tyDTMagToAGV2 ACCESS ADR(tyDTMagToAGV2);
//	p_tyDTMagToAGV3 ACCESS ADR(tyDTMagToAGV3);

END_ACTION
```

#### Act_Initial.st - Do Not Change!!!
```iecst
(** 2019-04-08 **)
ACTION Act_Initial:

	//Initial
	sStatTxt	:= a_sStatText[eStat];

	fbClntConnect.udiSndBffrSize		:= p_udiSndBffrSize;
	fbClntConnect.udiRcvBffrSize		:= p_udiRcvBffrSize;
	fbClntConnect.udiAliveIdleTmInSec	:= p_udiAliveIdleTimeInSec;
	fbClntConnect.tConnectTO			:= p_tConnTimeOut;
	fbClntConnect(bEn := FALSE);

	fbRcv.udiBffrSize	:= SIZEOF(sRcv);
	fbRcv.p_BffrDest	:= ADR(sRcv);
	fbRcv(bEn := FALSE);

	fbSend.p_BffrDest	:= ADR(sSnd);
	fbSend(bEn := FALSE);

	fbClose(bEn := FALSE);

	fbDirCreate1.sDevice	:= 'F';
	fbDirCreate1.sDirName	:= 'User';
	fbDirCreate1(bEn := FALSE);

	fbDirCreate2.sDevice	:= 'User';
	fbDirCreate2.sDirName	:= 'Log';
	fbDirCreate2(bEn := FALSE);

	fbFileAppend1.sDevice	:= 'Log';
	fbFileAppend1(bEn := FALSE);

	fbFileOldDel1.sDevice			:= 'Log';
	fbFileOldDel1.sPath				:= '';
	fbFileOldDel1.sKeyword			:= p_sProgNm;
	fbFileOldDel1.udiFileKeepDay	:= p_udiFileKeepDay;
	fbFileOldDel1(bEn := FALSE);

END_ACTION
```

#### Act_Main.st - Do Not Change!!!
```iecst
(** 2019-05-04 **)
ACTION Act_Main:
	//Set p_eAct
	IF eStatus = Idle OR eStatus = Busy OR eStatus = Done THEN
		eStat	:= p_eAct;
	END_IF

	IF eStatOld <> eStat THEN
		fbDirCreate1(bEn := FALSE);
		fbDirCreate2(bEn := FALSE);;
		usiStep			:= 0;

		sStatTxt	:= a_sStatText[eStat];

		eStatOld	:= eStat;

		eStatus		:= Busy;
	END_IF

	//Main
	CASE eStat OF

		TCPActIdle:
			eStatus	:= Idle;

		TCPActCreateDir:
			IF eStatus = Idle OR eStatus = Busy THEN

				eStatus	:= Busy;

				CASE usiStep OF
					0:
						fbDirCreate1(bEn := TRUE);
						IF fbDirCreate1.udiStatus = 0 THEN
							usiStep	:= 1;
						ELSIF fbDirCreate1.udiStatus < 65534 THEN
							eStatus		:= Error;

							IF fbDirCreate1.udiStatus = 1908 THEN
								udiStatus	:= 10016;	//Create User Directory Error
							ELSE
								udiStatus	:= fbDirCreate1.udiStatus;
							END_IF
						END_IF

					1:
						fbDirCreate2(bEn := TRUE);
						IF fbDirCreate2.udiStatus = 0 THEN
							eStatus	:= Done;
						ELSIF fbDirCreate2.udiStatus < 65534 THEN
							eStatus		:= Error;

							IF fbDirCreate2.udiStatus = 1908 THEN
								udiStatus	:= 10017;	//Create Log Directory Error
							ELSE
								udiStatus	:= fbDirCreate2.udiStatus;
							END_IF
						END_IF
				END_CASE

			END_IF

		TCPActDeleteOldLog:
			IF eStatus = Idle OR eStatus = Busy THEN

				eStatus	:= Busy;

				fbFileOldDel1.dtDTNow	:= p_dtCurrDT;
				fbFileOldDel1(bEn := TRUE);
				IF fbFileOldDel1.udiStatus = 0 THEN
					eStatus	:= Done;
				ELSIF fbFileOldDel1.udiStatus < 65534 THEN
					eStatus		:= Error;

					IF fbFileOldDel1.udiStatus = 1910 THEN
						udiStatus	:= 10154;	//Get Directory Info Error While Deleting Old Log
					ELSIF fbFileOldDel1.udiStatus = 1911 THEN
						udiStatus	:= 10155;	//Directory Read Error While Deleting Old Log
					ELSIF fbFileOldDel1.udiStatus = 1912 THEN
						udiStatus	:= 10156;	//File Delete Error While Deleting Old Log
					ELSE
						udiStatus	:= fbFileOldDel1.udiStatus;
					END_IF
				END_IF

			END_IF

		ELSE
			IF eStatus = Idle OR eStatus = Busy THEN
				eStatus	:= Done;
			END_IF

	END_CASE

END_ACTION
```

#### Act_Background.st - Do Not Change!!!
```iecst
(** 2019-06-10 **)
ACTION Act_Background:

	IF bRun = TRUE THEN
		IF eTCPModel = Client THEN
			IF udiTCPIdent = 0 THEN
				Act_Background_TCPConnect;
			ELSE
				IF bRstConnection = FALSE THEN
					Act_Background_TCPRcv;
					Act_Background_ChkAlive;
					Act_Background_TCPSend;
					Act_Background_TCPProcess;
			//		Act_Background_Log;
				ELSE
					Act_Background_TCPClose;
				END_IF
			END_IF
			Act_Background_Stop;

		ELSIF eTCPModel = Server THEN
			Act_TCPSvr;
			Act_TCPSvrProcess;
		END_IF

	END_IF

	IF EDGENEG(bRun) OR EDGENEG(udiTCPIdent = 0) THEN
		//Reset
		fbClntConnect(bEn := FALSE);

		bConnected		:= bRun;

		bWaitAliveResponse	:= FALSE;
		bCheckAliveTimeout 	:= FALSE;
	END_IF

	IF EDGENEG(bRun) OR EDGENEG(udiTCPIdent <> 0) THEN
		fbRcv(bEn := FALSE);

		fbSend(bEn := FALSE);
		fbClose(bEn := FALSE);

		fbFileAppend1(bEn := FALSE);
		iWriteLogStep	:= 0;

		bConnected		:= FALSE;

		memset(ADR(a_sMsgSend) , 0 , SIZEOF(a_sMsgSend));
		memset(ADR(tyAIVMsgRcvData) , 0 , SIZEOF(tyAIVMsgRcvData));
		udiMsgSendBffr	:= 0;
		bLoginSuccess 	:= FALSE;

		bWaitAliveResponse	:= FALSE;
		bCheckAliveTimeout 	:= FALSE;
	END_IF

	//Reset Error
	IF (eStatus1 = Error) AND bRstErr THEN
		eStatus1	:= Idle;
		udiStatus1	:= 0;

		fbClntConnect(bEn := FALSE);
		fbRcv(bEn := FALSE);
		fbSend(bEn := FALSE);
		fbClose(bEn := FALSE);

		fbFileAppend1(bEn := FALSE);
		iWriteLogStep	:= 0;

		bConnected		:= FALSE;

		memset(ADR(a_sMsgSend) , 0 , SIZEOF(a_sMsgSend));
		memset(ADR(tyAIVMsgRcvData) , 0 , SIZEOF(tyAIVMsgRcvData));
		udiMsgSendBffr	:= 0;
		bLoginSuccess 	:= FALSE;

		bWaitAliveResponse	:= FALSE;
		bCheckAliveTimeout 	:= FALSE;
	END_IF

	IF (eStatus2 = Error) AND bRstErr THEN
		eStatus2	:= Idle;
		udiStatus2	:= 0;

		fbFileAppend1(bEn := FALSE);
		iWriteLogStep	:= 0;

	END_IF

END_ACTION
```

#### Act_Background_ChkAlive.st - Do Not Change!!!
```iecst
(** 2019-05-30 **)
ACTION Act_Background_ChkAlive:

	fbSendAliveTimer.PT	:= T#30s;
	fbSendAliveTimer(IN:= bLoginSuccess);

	IF bWaitAliveResponse AND bCheckAliveTimeout=FALSE THEN

		fbCheckAliveTimer.PT	:= T#10s;
		fbCheckAliveTimer(IN:= TRUE);

		IF tyAIVMsgRcvData.bOneLineStatus THEN

			fbCheckAliveTimer(IN:= FALSE);
			bWaitAliveResponse	:= FALSE;
			bCheckAliveTimeout 	:= FALSE;

			tyAIVMsgRcvData.bOneLineStatus := FALSE;

			iFindBatteryLvl := FIND(sDecodeMsg, 'StateOfCharge:');

			IF iFindBatteryLvl <> 0 THEN

				sExtractBatteryLvl := MID(sDecodeMsg, 20 ,iFindBatteryLvl);
				sExtractBatteryLvl := RIGHT(sExtractBatteryLvl, 5);

				rCurrentBatteryLvl := STRING_TO_REAL(sExtractBatteryLvl);

			END_IF

		ELSIF fbCheckAliveTimer.Q THEN

			fbCheckAliveTimer(IN:= FALSE);
			bWaitAliveResponse	:= FALSE;
			bCheckAliveTimeout 	:= TRUE;

		END_IF
	END_IF

END_ACTION
```

#### Act_Background_TCPConnect.st - Do Not Change!!!
```iecst
(** 2020-09-10 **)
ACTION Act_Background_TCPConnect:

	IF eStatus1 <> Error THEN

		//Connect Server
		fbClntConnect.sClntIP		:= p_sIPAddr;
		fbClntConnect.sSvrIP		:= p_sSvrIP;
		fbClntConnect.uiClntPort	:= p_uiClientPort;
		fbClntConnect.uiSvrPort		:= p_uiSvrPort;
		fbClntConnect(bEn := TRUE);

		IF fbClntConnect.udiStatus = 0 THEN
			udiTCPIdent	:= fbClntConnect.udiTCPIdent;
			fbClntConnect(bEn := FALSE);

		ELSIF fbClntConnect.udiStatus = 2313 THEN
			fbClntConnect(bEn := FALSE);

		ELSIF fbClntConnect.udiStatus = 2323 OR bConnected= FALSE THEN
			udiStatus3	:= 10013;	//Client Connect Time Out // change to udistatus3
			//		udiStatus1	:= 10013;	//Client Connect Time Out

		ELSIF fbClntConnect.udiStatus < 65534 THEN
			eStatus1	:= Error;

			IF fbClntConnect.udiStatus = 2300 THEN
				udiStatus1	:= 10000;	//Invalid Ident While Client Connecting
			ELSIF fbClntConnect.udiStatus = 2302 THEN
				udiStatus1	:= 10001;	//Setting Keep Alive Interval Time Error While Client Connecting
			ELSIF fbClntConnect.udiStatus = 2303 THEN
				udiStatus1	:= 10002;	//Setting Keep Alive Idle Time Error While Client Connecting
			ELSIF fbClntConnect.udiStatus = 2304 THEN
				udiStatus1	:= 10003;	//Setting Keep Alive Count Error While Client Connecting
			ELSIF fbClntConnect.udiStatus = 2305 THEN
				udiStatus1	:= 10004;	//Setting Keep Alive Error While Client Connecting
			ELSIF fbClntConnect.udiStatus = 2306 THEN
				udiStatus1	:= 10005;	//Setting Receive Buffer Error While Client Connecting
			ELSIF fbClntConnect.udiStatus = 2307 THEN
				udiStatus1	:= 10006;	//Setting Send Buffer Error While Client Connecting
			ELSIF fbClntConnect.udiStatus = 2308 THEN
				udiStatus1	:= 10007;	//Setting No Waiting Error While Client Connecting
			ELSIF fbClntConnect.udiStatus = 2309 THEN
				udiStatus1	:= 10008;	//TCP Open Port Error While Client Connecting
			ELSIF fbClntConnect.udiStatus = 2310 THEN
				udiStatus1	:= 10009;	//Closing TCP Error While Client Connecting
			ELSIF fbClntConnect.udiStatus = 2313 THEN
				udiStatus1	:= 10010;	//Server Connection Failed While Client Connecting
			ELSIF fbClntConnect.udiStatus = 2314 THEN
				udiStatus1	:= 10011;	//Ident In Used While Client Connecting
			ELSIF fbClntConnect.udiStatus = 2315 THEN
				udiStatus1	:= 10012;	//Connect To Server Error While Client Connecting

			ELSE
				udiStatus1	:= fbClntConnect.udiStatus;
			END_IF

		END_IF

	END_IF

END_ACTION
```

#### Act_Background_TCPProcess.st - Do Not Change!!!
```iecst
(** 2019-06-10 **)
ACTION Act_Background_TCPProcess:

	IF tyAIVMsgRcvData.bEnterPW THEN

		a_sMsgSend[udiMsgSendBffr] := 'Hello$r$n';

		udiMsgSendBffr	:= udiMsgSendBffr + 1;

		tyAIVMsgRcvData.bEnterPW	:= FALSE;

	ELSIF tyAIVMsgRcvData.bLoginSuccess THEN

		bLoginSuccess := TRUE;

		tyAIVMsgRcvData.bLoginSuccess	:= FALSE;

		a_sMsgSend[udiMsgSendBffr]	:= 'qc status inprogress$r$nqc status pending$r$n';

		udiMsgSendBffr	:= udiMsgSendBffr + 1;

	ELSIF fbSendAliveTimer.Q THEN

		fbSendAliveTimer(IN:= FALSE);
		a_sMsgSend[udiMsgSendBffr] := 'onelinestatus$r$n';

		udiMsgSendBffr	:= udiMsgSendBffr + 1;

		bWaitAliveResponse := TRUE;

	ELSIF p_sMsgSnd <> ''  THEN

		a_sMsgSend[udiMsgSendBffr] := p_sMsgSnd;
		p_sMsgSnd	:= '';

		udiMsgSendBffr	:= udiMsgSendBffr + 1;
	END_IF

END_ACTION
```

#### Act_Background_TCPRcv.st - Do Not Change!!!
```iecst
(** 2019-06-10 **)
ACTION Act_Background_TCPRcv:

	IF eStatus1 <> Error THEN

		//Receive Data
		fbRcv.udiTCPIdent	:= udiTCPIdent;
		fbRcv(bEn := TRUE);

		IF (fbRcv.udiStatus = 0) OR (LEN(sRcv) > 0) THEN

			fLogDTConvert(ADR(sDT) , p_dtCurrDT);
			memset(ADR(a_sLogList[udiLogCntr]) , 0 , SIZEOF(a_sLogList[udiLogCntr]));
			memcpy(ADR(a_sLogList[udiLogCntr]) + LEN(a_sLogList[udiLogCntr]) , ADR(sDT) , LEN(sDT));
			memcpy(ADR(a_sLogList[udiLogCntr]) + LEN(a_sLogList[udiLogCntr]) , ADR('$r$n') , LEN('$r$n'));
			memcpy(ADR(a_sLogList[udiLogCntr]) + LEN(a_sLogList[udiLogCntr]) , ADR('RCV_FRM_AIV$r$n') , LEN('RCV_FRM_AIV$r$n'));
			memcpy(ADR(a_sLogList[udiLogCntr]) + LEN(a_sLogList[udiLogCntr]) , ADR(sRcv) , LEN(sRcv));
			memcpy(ADR(a_sLogList[udiLogCntr]) + LEN(a_sLogList[udiLogCntr]) , ADR('$r$n$r$n') , LEN('$r$n$r$n'));

			udiLogCntr	:= udiLogCntr + 1;
			IF udiLogCntr = 11 THEN
				udiLogCntr	:= 1;
			END_IF

			IF iHistoryCntr < 9 THEN
				a_tyHistoryList[iHistoryCntr].eTCP := MsgRcvFromTCP;
				a_tyHistoryList[iHistoryCntr].sMsg := sRcv;
				iHistoryCntr := iHistoryCntr +1 ;
			ELSE
				memmove(ADR(a_tyHistoryList[1]),ADR(a_tyHistoryList[2]),(SIZEOF(a_tyHistoryList[1])*7));
				memset(ADR(a_tyHistoryList[8]),0,SIZEOF(a_tyHistoryList[1]));
				a_tyHistoryList[8].eTCP := MsgRcvFromTCP;
				a_tyHistoryList[8].sMsg := sRcv;
			END_IF

			IF FIND(sRcv , 'Enter password') <> 0 THEN
				tyAIVMsgRcvData.bEnterPW	:= TRUE;

			ELSIF FIND(sRcv , sELD1Reached) <> 0 THEN
				tyAIVMsgRcvData.bELD1Reached	:= TRUE;

			ELSIF FIND(sRcv , sELD1Completed) <> 0 THEN
				tyAIVMsgRcvData.bELD1Completed	:= TRUE;

			ELSIF FIND(sRcv , sELD2Reached) <> 0 THEN
				tyAIVMsgRcvData.bELD2Reached	:= TRUE;

			ELSIF FIND(sRcv , sELD2Completed) <> 0 THEN
				tyAIVMsgRcvData.bELD2Completed	:= TRUE;

			ELSIF FIND(sRcv , sELD3Reached) <> 0 THEN
				tyAIVMsgRcvData.bELD3Reached	:= TRUE;

			ELSIF FIND(sRcv , sELD3Completed) <> 0 THEN
				tyAIVMsgRcvData.bELD3Completed	:= TRUE;

			ELSIF FIND(sRcv , sEUL1Reached) <> 0 THEN
				tyAIVMsgRcvData.bEUL1Reached	:= TRUE;

			ELSIF FIND(sRcv , sEUL1Completed) <> 0 THEN
				tyAIVMsgRcvData.bEUL1Completed	:= TRUE;

			ELSIF FIND(sRcv , sEUL2Reached) <> 0 THEN
				tyAIVMsgRcvData.bEUL2Reached	:= TRUE;

			ELSIF FIND(sRcv , sEUL2Completed) <> 0 THEN
				tyAIVMsgRcvData.bEUL2Completed	:= TRUE;

			ELSIF FIND(sRcv , sEUL3Reached) <> 0 THEN
				tyAIVMsgRcvData.bEUL3Reached	:= TRUE;

			ELSIF FIND(sRcv , sEUL3Completed) <> 0 THEN
				tyAIVMsgRcvData.bEUL3Completed	:= TRUE;

			ELSIF FIND(sRcv , sSTANDBYReached) <> 0 THEN
				tyAIVMsgRcvData.bStandbyReached	:= TRUE;

			ELSIF FIND(sRcv , sSTANDBYCompleted) <> 0 THEN
				tyAIVMsgRcvData.bStandbyCompleted	:= TRUE;

			ELSIF FIND(sRcv, 'Arrived at clear') <> 0 THEN
				tyAIVMsgRcvData.bMoveBackCompleted	:= TRUE;

			ELSIF FIND(sRcv, 'Status:') <> 0 THEN
				tyAIVMsgRcvData.bOneLineStatus	:= TRUE;

				sDecodeMsg := sRcv;

			ELSIF FIND(sRcv, 'Welcome to the server') <> 0 THEN
				tyAIVMsgRcvData.bLoginSuccess	:= TRUE;

			END_IF

			fbRcv(bEn := FALSE);

			memset(ADR(sRcv) , 0 , SIZEOF(sRcv));

		ELSIF (fbRcv.udiStatus = 2317)  THEN
			fbRcv(bEn := FALSE);

			memset(ADR(sRcv) , 0 , SIZEOF(sRcv));

		ELSIF (fbRcv.udiStatus = 2316)  THEN
			bRstConnection	:= TRUE;

			memset(ADR(sRcv) , 0 , SIZEOF(sRcv));

		ELSIF (fbRcv.udiStatus = 2318)  THEN
			bRstConnection	:= TRUE;

			memset(ADR(sRcv) , 0 , SIZEOF(sRcv));

		ELSIF (fbRcv.udiStatus < 65534)  THEN
			eStatus1	:= Error;

			IF fbRcv.udiStatus = 2300 THEN
				udiStatus1	:= 10014;	//Invalid Ident While Receiving Data
			ELSIF fbRcv.udiStatus = 2319 THEN
				udiStatus1	:= 10015;	//TCP Receive Data Error While Receiving Data
			ELSE
				udiStatus1	:= fbRcv.udiStatus;
			END_IF

			memset(ADR(sRcv) , 0 , SIZEOF(sRcv));

		END_IF

	END_IF

END_ACTION
```

#### Act_Background_TCPSend.st - Do Not Change!!!
```iecst
(** 2019-06-10 **)
ACTION Act_Background_TCPSend:

	//Message Send (Generate XML Message)
	IF a_sMsgSend[0] <> '' THEN

		memset(ADR(sSnd) , 0 , SIZEOF(sSnd));

		sSnd			:= a_sMsgSend[0];
		udiSndMsgLen	:= LEN(sSnd);

		//Message Send
		fbSend.udiTCPIdent	:= udiTCPIdent;
		fbSend.udiSndSize	:= udiSndMsgLen;
		fbSend(bEn := TRUE);

		IF (fbSend.udiStatus = 0) THEN

			fLogDTConvert(ADR(sDT) , p_dtCurrDT);
			memset(ADR(a_sLogList[udiLogCntr]) , 0 , SIZEOF(a_sLogList[udiLogCntr]));
			memcpy(ADR(a_sLogList[udiLogCntr]) + LEN(a_sLogList[udiLogCntr]) , ADR(sDT) , LEN(sDT));
			memcpy(ADR(a_sLogList[udiLogCntr]) + LEN(a_sLogList[udiLogCntr]) , ADR('$r$n') , LEN('$r$n'));
			memcpy(ADR(a_sLogList[udiLogCntr]) + LEN(a_sLogList[udiLogCntr]) , ADR('SND_TO_AIV$r$n') , LEN('SND_TO_AIV$r$n'));
			memcpy(ADR(a_sLogList[udiLogCntr]) + LEN(a_sLogList[udiLogCntr]) , ADR(sSnd) , LEN(sSnd));
			memcpy(ADR(a_sLogList[udiLogCntr]) + LEN(a_sLogList[udiLogCntr]) , ADR('$r$n$r$n') , LEN('$r$n$r$n'));

			udiLogCntr	:= udiLogCntr + 1;
			IF udiLogCntr = 11 THEN
				udiLogCntr	:= 1;
			END_IF

			IF iHistoryCntr < 9 THEN
				a_tyHistoryList[iHistoryCntr].eTCP := MsgSndToTCP;
				a_tyHistoryList[iHistoryCntr].sMsg := sSnd;
				iHistoryCntr := iHistoryCntr +1 ;
			ELSE
				memmove(ADR(a_tyHistoryList[1]),ADR(a_tyHistoryList[2]),(SIZEOF(a_tyHistoryList[1])*7));
				memset(ADR(a_tyHistoryList[8]),0,SIZEOF(a_tyHistoryList[1]));
				a_tyHistoryList[8].eTCP := MsgSndToTCP;
				a_tyHistoryList[8].sMsg := sSnd;
			END_IF

			memcpy(ADR(a_sMsgSend[0]) , ADR(a_sMsgSend[1]) , SIZEOF(a_sMsgSend[0]) * 50);
			a_sMsgSend[50]		:= '';
			udiMsgSendBffr		:= udiMsgSendBffr - 1;

			fbSend(bEn := FALSE);

		ELSIF (fbSend.udiStatus = 2321)  THEN
			bRstConnection	:= TRUE;

		ELSIF (fbSend.udiStatus < 65534)  THEN
			eStatus1	:= Error;

			IF fbSend.udiStatus = 2300 THEN
				udiStatus1	:= 10024;	//Invalid Ident While Sending Data
			ELSIF fbSend.udiStatus = 2320 THEN
				udiStatus1	:= 10025;	//TCP Retry Send Data Error While Sending Data
			ELSIF fbSend.udiStatus = 2322 THEN
				udiStatus1	:= 10026;	//TCP Send Data Error
			ELSE
				udiStatus1	:= fbSend.udiStatus;
			END_IF

		END_IF

	END_IF

END_ACTION
```
